LIN {X 0,Y 361.833,Z 229.413,A -85,B 0,C 180,E1 -13010.986,E2 -13010.986} C_VEL
LIN {X 0,Y 361.881,Z 229.41,A -85,B 0,C 180,E1 -13014.66,E2 -13014.66} C_VEL
LIN {X 0,Y 361.859,Z 229.412,A -85,B 0,C 180,E1 -13017.057,E2 -13017.057} C_VEL
LIN {X 0,Y 361.93,Z 229.564,A -85,B 0,C 180,E1 -13019.451,E2 -13019.451} C_VEL
LIN {X 0,Y 364.526,Z 241.261,A -85,B 0,C 180,E1 -13022.49,E2 -13022.49} C_VEL
LIN {X 0,Y 366.114,Z 250.204,A -85,B 0,C 180,E1 -13024.69,E2 -13024.69} C_VEL
LIN {X 0,Y 364.917,Z 262.619,A -85,B 0,C 180,E1 -13027.439,E2 -13027.439} C_VEL
LIN {X 0,Y 368.835,Z 283.762,A -85,B 0,C 180,E1 -13028.191,E2 -13028.191} C_VEL
LIN {X 0,Y 370.98,Z 298.524,A -85,B 0,C 180,E1 -13028.66,E2 -13028.66} C_VEL
LIN {X 0,Y 369.479,Z 372.16,A -85,B 0,C 180,E1 -13030.196,E2 -13030.196} C_VEL
LIN {X 0,Y 368.702,Z 385.754,A -85,B 0,C 180,E1 -13030.696,E2 -13030.696} C_VEL
LIN {X 0,Y 367.704,Z 398.62,A -85,B 0,C 180,E1 -13031.401,E2 -13031.401} C_VEL
LIN {X 0,Y 366.629,Z 410.378,A -85,B 0,C 180,E1 -13032.284,E2 -13032.284} C_VEL
LIN {X 0,Y 365.424,Z 421.749,A -85,B 0,C 180,E1 -13033.377,E2 -13033.377} C_VEL
LIN {X 0,Y 364.348,Z 431.632,A -85,B 0,C 180,E1 -13034.565,E2 -13034.565} C_VEL
LIN {X 0,Y 363.296,Z 441.299,A -85,B 0,C 180,E1 -13036.007,E2 -13036.007} C_VEL
LIN {X 0,Y 362.237,Z 450.344,A -85,B 0,C 180,E1 -13037.678,E2 -13037.678} C_VEL
LIN {X 0,Y 361.437,Z 457.643,A -85,B 0,C 180,E1 -13039.355,E2 -13039.355} C_VEL
LIN {X 0,Y 360.913,Z 463.485,A -85,B 0,C 180,E1 -13041.038,E2 -13041.038} C_VEL
LIN {X 0,Y 360.54,Z 468.095,A -85,B 0,C 180,E1 -13042.721,E2 -13042.721} C_VEL
LIN {X 0,Y 360.346,Z 471.611,A -85,B 0,C 180,E1 -13044.404,E2 -13044.404} C_VEL
LIN {X 0,Y 360.346,Z 473.371,A -85,B 0,C 180,E1 -13045.526,E2 -13045.526} C_VEL
LIN {X 0,Y 360.306,Z 474.719,A -85,B 0,C 180,E1 -13046.645,E2 -13046.645} C_VEL
LIN {X 0,Y 360.305,Z 475.671,A -85,B 0,C 180,E1 -13047.764,E2 -13047.764} C_VEL
LIN {X 0,Y 360.353,Z 476.208,A -85,B 0,C 180,E1 -13048.883,E2 -13048.883} C_VEL
LIN {X 0,Y 360.404,Z 476.312,A -85,B 0,C 180,E1 -13050,E2 -13050} C_VEL
LIN {X 0,Y 360.368,Z 476.021,A -85,B 0,C 180,E1 -13051.118,E2 -13051.118} C_VEL
LIN {X 0,Y 360.309,Z 475.335,A -85,B 0,C 180,E1 -13052.236,E2 -13052.236} C_VEL
LIN {X 0,Y 360.311,Z 474.232,A -85,B 0,C 180,E1 -13053.355,E2 -13053.355} C_VEL
LIN {X 0,Y 360.368,Z 472.675,A -85,B 0,C 180,E1 -13054.474,E2 -13054.474} C_VEL
LIN {X 0,Y 360.395,Z 469.967,A -85,B 0,C 180,E1 -13055.961,E2 -13055.961} C_VEL
LIN {X 0,Y 360.636,Z 465.301,A -85,B 0,C 180,E1 -13057.84,E2 -13057.84} C_VEL
LIN {X 0,Y 361.085,Z 458.852,A -85,B 0,C 180,E1 -13059.805,E2 -13059.805} C_VEL
LIN {X 0,Y 361.659,Z 451.801,A -85,B 0,C 180,E1 -13061.489,E2 -13061.489} C_VEL
LIN {X 0,Y 362.587,Z 442.961,A -85,B 0,C 180,E1 -13063.164,E2 -13063.164} C_VEL
LIN {X 0,Y 363.61,Z 432.861,A -85,B 0,C 180,E1 -13064.703,E2 -13064.703} C_VEL
LIN {X 0,Y 364.434,Z 422.644,A -85,B 0,C 180,E1 -13065.95,E2 -13065.95} C_VEL
LIN {X 0,Y 365.491,Z 411.272,A -85,B 0,C 180,E1 -13067.052,E2 -13067.052} C_VEL
LIN {X 0,Y 366.457,Z 399.49,A -85,B 0,C 180,E1 -13067.941,E2 -13067.941} C_VEL
LIN {X 0,Y 367.363,Z 386.617,A -85,B 0,C 180,E1 -13068.653,E2 -13068.653} C_VEL
LIN {X 0,Y 367.996,Z 374.094,A -85,B 0,C 180,E1 -13069.126,E2 -13069.126} C_VEL
LIN {X 0,Y 368.512,Z 346.999,A -85,B 0,C 180,E1 -13069.713,E2 -13069.713} C_VEL
LIN {X 0,Y 369.284,Z 296.844,A -85,B 0,C 180,E1 -13070.734,E2 -13070.734} C_VEL
LIN {X 0,Y 364.271,Z 263.791,A -85,B 0,C 180,E1 -13071.746,E2 -13071.746} C_VEL
LIN {X 0,Y 365.634,Z 249.234,A -85,B 0,C 180,E1 -13075.015,E2 -13075.015} C_VEL
LIN {X 0,Y 364.83,Z 243.927,A -85,B 0,C 180,E1 -13076.299,E2 -13076.299} C_VEL
LIN {X 0,Y 362.103,Z 230.432,A -85,B 0,C 180,E1 -13079.699,E2 -13079.699} C_VEL
LIN {X 0,Y 361.875,Z 229.413,A -85,B 0,C 180,E1 -13080.023,E2 -13080.023} C_VEL
LIN {X 0,Y 361.845,Z 229.41,A -85,B 0,C 180,E1 -13083.36,E2 -13083.36} C_VEL
LIN {X 0,Y 361.867,Z 229.406,A -85,B 0,C 180,E1 -13087.017,E2 -13087.017} C_VEL
LIN {X 0,Y 361.814,Z 229.412,A -85,B 0,C 180,E1 -13090.746,E2 -13090.746} C_VEL
LIN {X 0,Y 361.785,Z 229.417,A -85,B 0,C 180,E1 -13094.372,E2 -13094.372} C_VEL
LIN {X 0,Y 361.816,Z 229.417,A -85,B 0,C 180,E1 -13097.57,E2 -13097.57} C_VEL
LIN {X 0,Y 361.83,Z 229.411,A -85,B 0,C 180,E1 -13100.979,E2 -13100.979} C_VEL
LIN {X 0,Y 361.874,Z 229.405,A -85,B 0,C 180,E1 -13104.653,E2 -13104.653} C_VEL
LIN {X 0,Y 361.852,Z 229.408,A -85,B 0,C 180,E1 -13107.05,E2 -13107.05} C_VEL
LIN {X 0,Y 361.856,Z 229.408,A -85,B 0,C 180,E1 -13110.946,E2 -13110.946} C_VEL
LIN {X 0,Y 361.869,Z 229.405,A -85,B 0,C 180,E1 -13114.7,E2 -13114.7} C_VEL
LIN {X 0,Y 361.862,Z 229.407,A -85,B 0,C 180,E1 -13118.34,E2 -13118.34} C_VEL
LIN {X 0,Y 361.906,Z 229.403,A -85,B 0,C 180,E1 -13122.087,E2 -13122.087} C_VEL
LIN {X 0,Y 361.958,Z 229.398,A -85,B 0,C 180,E1 -13125.374,E2 -13125.374} C_VEL
LIN {X 0,Y 361.956,Z 229.395,A -85,B 0,C 180,E1 -13128.798,E2 -13128.798} C_VEL
LIN {X 0,Y 362.072,Z 229.381,A -85,B 0,C 180,E1 -13132.185,E2 -13132.185} C_VEL
LIN {X 0,Y 362.079,Z 229.379,A -85,B 0,C 180,E1 -13134.425,E2 -13134.425} C_VEL
LIN {X 0,Y 362.245,Z 229.362,A -85,B 0,C 180,E1 -13137.77,E2 -13137.77} C_VEL
LIN {X 0,Y 362.255,Z 229.358,A -85,B 0,C 180,E1 -13142.217,E2 -13142.217} C_VEL
LIN {X 0,Y 362.1,Z 229.377,A -85,B 0,C 180,E1 -13146.681,E2 -13146.681} C_VEL
LIN {X 0,Y 361.979,Z 229.393,A -85,B 0,C 180,E1 -13150.056,E2 -13150.056} C_VEL
LIN {X 0,Y 361.979,Z 229.394,A -85,B 0,C 180,E1 -13153.892,E2 -13153.892} C_VEL
LIN {X 0,Y 361.905,Z 229.403,A -85,B 0,C 180,E1 -13156.928,E2 -13156.928} C_VEL
LIN {X 0,Y 361.869,Z 229.405,A -85,B 0,C 180,E1 -13160.454,E2 -13160.454} C_VEL
LIN {X 0,Y 361.866,Z 229.406,A -85,B 0,C 180,E1 -13164.106,E2 -13164.106} C_VEL
LIN {X 0,Y 361.853,Z 229.41,A -85,B 0,C 180,E1 -13167.775,E2 -13167.775} C_VEL
LIN {X 0,Y 361.814,Z 229.418,A -85,B 0,C 180,E1 -13171.279,E2 -13171.279} C_VEL
LIN {X 0,Y 361.818,Z 229.412,A -85,B 0,C 180,E1 -13174.274,E2 -13174.274} C_VEL
LIN {X 0,Y 361.825,Z 229.416,A -85,B 0,C 180,E1 -13177.217,E2 -13177.217} C_VEL
LIN {X 0,Y 361.794,Z 229.416,A -85,B 0,C 180,E1 -13180.749,E2 -13180.749} C_VEL
LIN {X 0,Y 361.776,Z 229.417,A -85,B 0,C 180,E1 -13184.363,E2 -13184.363} C_VEL
LIN {X 0,Y 361.789,Z 229.419,A -85,B 0,C 180,E1 -13187.563,E2 -13187.563} C_VEL
LIN {X 0,Y 361.821,Z 229.415,A -85,B 0,C 180,E1 -13190.969,E2 -13190.969} C_VEL
LIN {X 0,Y 361.824,Z 229.412,A -85,B 0,C 180,E1 -13194.651,E2 -13194.651} C_VEL
LIN {X 0,Y 361.785,Z 229.416,A -85,B 0,C 180,E1 -13198.366,E2 -13198.366} C_VEL
LIN {X 0,Y 361.848,Z 229.412,A -85,B 0,C 180,E1 -13200.951,E2 -13200.951} C_VEL
LIN {X 0,Y 361.899,Z 229.405,A -85,B 0,C 180,E1 -13203.471,E2 -13203.471} C_VEL
LIN {X 0,Y 361.863,Z 229.413,A -85,B 0,C 180,E1 -13207.143,E2 -13207.143} C_VEL
LIN {X 0,Y 361.877,Z 229.407,A -85,B 0,C 180,E1 -13210.722,E2 -13210.722} C_VEL
LIN {X 0,Y 361.889,Z 229.403,A -85,B 0,C 180,E1 -13214.224,E2 -13214.224} C_VEL
LIN {X 0,Y 361.94,Z 229.398,A -85,B 0,C 180,E1 -13216.526,E2 -13216.526} C_VEL
LIN {X 0,Y 361.977,Z 229.392,A -85,B 0,C 180,E1 -13219.937,E2 -13219.937} C_VEL
LIN {X 0,Y 362.097,Z 229.377,A -85,B 0,C 180,E1 -13222.192,E2 -13222.192} C_VEL
LIN {X 0,Y 362.068,Z 229.381,A -85,B 0,C 180,E1 -13224.431,E2 -13224.431} C_VEL
LIN {X 0,Y 362.228,Z 229.361,A -85,B 0,C 180,E1 -13227.776,E2 -13227.776} C_VEL
LIN {X 0,Y 362.368,Z 229.343,A -85,B 0,C 180,E1 -13230,E2 -13230} C_VEL
LIN {X 0,Y 362.228,Z 229.361,A -85,B 0,C 180,E1 -13232.224,E2 -13232.224} C_VEL
LIN {X 0,Y 362.121,Z 229.377,A -85,B 0,C 180,E1 -13236.687,E2 -13236.687} C_VEL
LIN {X 0,Y 362.073,Z 229.567,A -85,B 0,C 180,E1 -13238.789,E2 -13238.789} C_VEL
LIN {X 0,Y 363.761,Z 238.743,A -85,B 0,C 180,E1 -13241.316,E2 -13241.316} C_VEL
LIN {X 0,Y 366.817,Z 248.552,A -85,B 0,C 180,E1 -13241.71,E2 -13241.71} C_VEL
LIN {X 0,Y 369.824,Z 264.217,A -85,B 0,C 180,E1 -13242.212,E2 -13242.212} C_VEL
LIN {X 0,Y 368.227,Z 346.682,A -85,B 0,C 180,E1 -13243.903,E2 -13243.903} C_VEL
LIN {X 0,Y 367.706,Z 359.685,A -85,B 0,C 180,E1 -13244.387,E2 -13244.387} C_VEL
LIN {X 0,Y 367.117,Z 371.772,A -85,B 0,C 180,E1 -13245.048,E2 -13245.048} C_VEL
LIN {X 0,Y 366.274,Z 384.403,A -85,B 0,C 180,E1 -13245.988,E2 -13245.988} C_VEL
LIN {X 0,Y 365.338,Z 395.535,A -85,B 0,C 180,E1 -13247.059,E2 -13247.059} C_VEL
LIN {X 0,Y 364.31,Z 406.448,A -85,B 0,C 180,E1 -13248.378,E2 -13248.378} C_VEL
LIN {X 0,Y 363.312,Z 415.93,A -85,B 0,C 180,E1 -13249.815,E2 -13249.815} C_VEL
LIN {X 0,Y 362.472,Z 424.801,A -85,B 0,C 180,E1 -13251.485,E2 -13251.485} C_VEL
LIN {X 0,Y 361.737,Z 431.855,A -85,B 0,C 180,E1 -13253.142,E2 -13253.142} C_VEL
LIN {X 0,Y 361.542,Z 433.936,A -85,B 0,C 180,E1 -13253.715,E2 -13253.715} C_VEL
LIN {X 0,Y 360.709,Z 436.714,A -85,B 0,C 180,E1 -13254.533,E2 -13254.533} C_VEL
LIN {X 0,Y 357.552,Z 440.748,A -85,B 0,C 180,E1 -13255.885,E2 -13255.885} C_VEL
LIN {X 0,Y 354.887,Z 443.525,A -85,B 0,C 180,E1 -13257.011,E2 -13257.011} C_VEL
LIN {X 0,Y 353.665,Z 445.304,A -85,B 0,C 180,E1 -13257.907,E2 -13257.907} C_VEL
LIN {X 0,Y 353.522,Z 445.8,A -85,B 0,C 180,E1 -13258.215,E2 -13258.215} C_VEL
LIN {X 0,Y 353.225,Z 448.061,A -85,B 0,C 180,E1 -13259.828,E2 -13259.828} C_VEL
LIN {X 0,Y 353.063,Z 449.259,A -85,B 0,C 180,E1 -13261.167,E2 -13261.167} C_VEL
LIN {X 0,Y 353.03,Z 450.068,A -85,B 0,C 180,E1 -13263.284,E2 -13263.284} C_VEL
LIN {X 0,Y 353.12,Z 449.518,A -85,B 0,C 180,E1 -13265.329,E2 -13265.329} C_VEL
LIN {X 0,Y 353.37,Z 447.743,A -85,B 0,C 180,E1 -13267.309,E2 -13267.309} C_VEL
LIN {X 0,Y 353.82,Z 444.396,A -85,B 0,C 180,E1 -13269.465,E2 -13269.465} C_VEL
LIN {X 0,Y 354.385,Z 439.268,A -85,B 0,C 180,E1 -13271.676,E2 -13271.676} C_VEL
LIN {X 0,Y 355.052,Z 434.218,A -85,B 0,C 180,E1 -13273.312,E2 -13273.312} C_VEL
LIN {X 0,Y 355.855,Z 428.017,A -85,B 0,C 180,E1 -13274.927,E2 -13274.927} C_VEL
LIN {X 0,Y 356.738,Z 421.001,A -85,B 0,C 180,E1 -13276.42,E2 -13276.42} C_VEL
LIN {X 0,Y 357.944,Z 411.554,A -85,B 0,C 180,E1 -13278.05,E2 -13278.05} C_VEL
LIN {X 0,Y 359.069,Z 402.36,A -85,B 0,C 180,E1 -13279.326,E2 -13279.326} C_VEL
LIN {X 0,Y 360.134,Z 392.431,A -85,B 0,C 180,E1 -13280.447,E2 -13280.447} C_VEL
LIN {X 0,Y 361.277,Z 380.527,A -85,B 0,C 180,E1 -13281.512,E2 -13281.512} C_VEL
LIN {X 0,Y 362.175,Z 368.681,A -85,B 0,C 180,E1 -13282.326,E2 -13282.326} C_VEL
LIN {X 0,Y 362.825,Z 356.306,A -85,B 0,C 180,E1 -13282.943,E2 -13282.943} C_VEL
LIN {X 0,Y 363.321,Z 342.566,A -85,B 0,C 180,E1 -13283.379,E2 -13283.379} C_VEL
LIN {X 0,Y 365.083,Z 265.657,A -85,B 0,C 180,E1 -13284.987,E2 -13284.987} C_VEL
LIN {X 0,Y 362.139,Z 252.353,A -85,B 0,C 180,E1 -13285.508,E2 -13285.508} C_VEL
LIN {X 0,Y 356.864,Z 239.401,A -85,B 0,C 180,E1 -13286.239,E2 -13286.239} C_VEL
LIN {X 0,Y 354.823,Z 230.291,A -85,B 0,C 180,E1 -13288.821,E2 -13288.821} C_VEL
LIN {X 0,Y 354.822,Z 230.288,A -85,B 0,C 180,E1 -13291.626,E2 -13291.626} C_VEL
LIN {X 0,Y 354.87,Z 230.279,A -85,B 0,C 180,E1 -13294.179,E2 -13294.179} C_VEL
LIN {X 0,Y 354.808,Z 230.287,A -85,B 0,C 180,E1 -13297.901,E2 -13297.901} C_VEL
LIN {X 0,Y 354.899,Z 230.279,A -85,B 0,C 180,E1 -13301.898,E2 -13301.898} C_VEL
LIN {X 0,Y 354.923,Z 230.272,A -85,B 0,C 180,E1 -13305.988,E2 -13305.988} C_VEL
LIN {X 0,Y 354.962,Z 230.269,A -85,B 0,C 180,E1 -13309.743,E2 -13309.743} C_VEL
LIN {X 0,Y 355.091,Z 230.254,A -85,B 0,C 180,E1 -13313.187,E2 -13313.187} C_VEL
LIN {X 0,Y 355.23,Z 230.231,A -85,B 0,C 180,E1 -13317.739,E2 -13317.739} C_VEL
LIN {X 0,Y 355.342,Z 230.22,A -85,B 0,C 180,E1 -13320.006,E2 -13320.006} C_VEL
LIN {X 0,Y 355.219,Z 230.23,A -85,B 0,C 180,E1 -13322.274,E2 -13322.274} C_VEL
LIN {X 0,Y 355.099,Z 230.248,A -85,B 0,C 180,E1 -13326.826,E2 -13326.826} C_VEL
LIN {X 0,Y 354.95,Z 230.263,A -85,B 0,C 180,E1 -13330.271,E2 -13330.271} C_VEL
LIN {X 0,Y 354.942,Z 230.266,A -85,B 0,C 180,E1 -13334.024,E2 -13334.024} C_VEL
LIN {X 0,Y 354.891,Z 230.273,A -85,B 0,C 180,E1 -13338.097,E2 -13338.097} C_VEL
LIN {X 0,Y 354.808,Z 230.284,A -85,B 0,C 180,E1 -13342.113,E2 -13342.113} C_VEL
LIN {X 0,Y 354.802,Z 230.285,A -85,B 0,C 180,E1 -13345.84,E2 -13345.84} C_VEL
LIN {X 0,Y 354.799,Z 230.285,A -85,B 0,C 180,E1 -13349.689,E2 -13349.689} C_VEL
LIN {X 0,Y 354.815,Z 230.281,A -85,B 0,C 180,E1 -13353.706,E2 -13353.706} C_VEL
LIN {X 0,Y 354.799,Z 230.287,A -85,B 0,C 180,E1 -13356.465,E2 -13356.465} C_VEL
LIN {X 0,Y 354.778,Z 230.289,A -85,B 0,C 180,E1 -13359.417,E2 -13359.417} C_VEL
LIN {X 0,Y 354.776,Z 230.295,A -85,B 0,C 180,E1 -13362.867,E2 -13362.867} C_VEL
LIN {X 0,Y 354.747,Z 230.302,A -85,B 0,C 180,E1 -13366.102,E2 -13366.102} C_VEL
LIN {X 0,Y 354.772,Z 230.293,A -85,B 0,C 180,E1 -13369.178,E2 -13369.178} C_VEL
LIN {X 0,Y 354.809,Z 230.289,A -85,B 0,C 180,E1 -13372.408,E2 -13372.408} C_VEL
LIN {X 0,Y 354.819,Z 230.288,A -85,B 0,C 180,E1 -13374.943,E2 -13374.943} C_VEL
LIN {X 0,Y 354.84,Z 230.387,A -85,B 0,C 180,E1 -13378.979,E2 -13378.979} C_VEL
LIN {X 0,Y 357.27,Z 241.039,A -85,B 0,C 180,E1 -13381.829,E2 -13381.829} C_VEL
LIN {X 0,Y 359.071,Z 250.386,A -85,B 0,C 180,E1 -13384.211,E2 -13384.211} C_VEL
LIN {X 0,Y 359.015,Z 254.237,A -85,B 0,C 180,E1 -13385.111,E2 -13385.111} C_VEL
LIN {X 0,Y 358.177,Z 262.294,A -85,B 0,C 180,E1 -13386.925,E2 -13386.925} C_VEL
LIN {X 0,Y 362.326,Z 284.308,A -85,B 0,C 180,E1 -13387.745,E2 -13387.745} C_VEL
LIN {X 0,Y 364.427,Z 299.076,A -85,B 0,C 180,E1 -13388.23,E2 -13388.23} C_VEL
LIN {X 0,Y 362.884,Z 372.032,A -85,B 0,C 180,E1 -13389.783,E2 -13389.783} C_VEL
LIN {X 0,Y 362.068,Z 385.57,A -85,B 0,C 180,E1 -13390.291,E2 -13390.291} C_VEL
LIN {X 0,Y 361.096,Z 397.89,A -85,B 0,C 180,E1 -13390.974,E2 -13390.974} C_VEL
LIN {X 0,Y 359.88,Z 410.544,A -85,B 0,C 180,E1 -13391.94,E2 -13391.94} C_VEL
LIN {X 0,Y 358.637,Z 421.837,A -85,B 0,C 180,E1 -13393.053,E2 -13393.053} C_VEL
LIN {X 0,Y 357.529,Z 431.546,A -85,B 0,C 180,E1 -13394.248,E2 -13394.248} C_VEL
LIN {X 0,Y 356.375,Z 441.257,A -85,B 0,C 180,E1 -13395.729,E2 -13395.729} C_VEL
LIN {X 0,Y 355.281,Z 450.253,A -85,B 0,C 180,E1 -13397.433,E2 -13397.433} C_VEL
LIN {X 0,Y 354.399,Z 457.509,A -85,B 0,C 180,E1 -13399.141,E2 -13399.141} C_VEL
LIN {X 0,Y 353.867,Z 463.313,A -85,B 0,C 180,E1 -13400.858,E2 -13400.858} C_VEL
LIN {X 0,Y 353.485,Z 467.901,A -85,B 0,C 180,E1 -13402.575,E2 -13402.575} C_VEL
LIN {X 0,Y 353.259,Z 471.4,A -85,B 0,C 180,E1 -13404.291,E2 -13404.291} C_VEL
LIN {X 0,Y 353.259,Z 473.149,A -85,B 0,C 180,E1 -13405.436,E2 -13405.436} C_VEL
LIN {X 0,Y 353.227,Z 474.49,A -85,B 0,C 180,E1 -13406.578,E2 -13406.578} C_VEL
LIN {X 0,Y 353.211,Z 475.432,A -85,B 0,C 180,E1 -13407.719,E2 -13407.719} C_VEL
LIN {X 0,Y 353.254,Z 475.95,A -85,B 0,C 180,E1 -13408.86,E2 -13408.86} C_VEL
LIN {X 0,Y 353.309,Z 476.044,A -85,B 0,C 180,E1 -13410,E2 -13410} C_VEL
LIN {X 0,Y 353.27,Z 475.742,A -85,B 0,C 180,E1 -13411.14,E2 -13411.14} C_VEL
LIN {X 0,Y 353.215,Z 475.047,A -85,B 0,C 180,E1 -13412.281,E2 -13412.281} C_VEL
LIN {X 0,Y 353.232,Z 473.922,A -85,B 0,C 180,E1 -13413.422,E2 -13413.422} C_VEL
LIN {X 0,Y 353.28,Z 472.353,A -85,B 0,C 180,E1 -13414.564,E2 -13414.564} C_VEL
LIN {X 0,Y 353.351,Z 469.184,A -85,B 0,C 180,E1 -13416.28,E2 -13416.28} C_VEL
LIN {X 0,Y 353.568,Z 464.928,A -85,B 0,C 180,E1 -13417.998,E2 -13417.998} C_VEL
LIN {X 0,Y 354.043,Z 458.448,A -85,B 0,C 180,E1 -13420.002,E2 -13420.002} C_VEL
LIN {X 0,Y 354.667,Z 451.351,A -85,B 0,C 180,E1 -13421.719,E2 -13421.719} C_VEL
LIN {X 0,Y 355.599,Z 442.465,A -85,B 0,C 180,E1 -13423.428,E2 -13423.428} C_VEL
LIN {X 0,Y 356.601,Z 433.359,A -85,B 0,C 180,E1 -13424.845,E2 -13424.845} C_VEL
LIN {X 0,Y 357.446,Z 423.303,A -85,B 0,C 180,E1 -13426.124,E2 -13426.124} C_VEL
LIN {X 0,Y 358.549,Z 412.143,A -85,B 0,C 180,E1 -13427.245,E2 -13427.245} C_VEL
LIN {X 0,Y 359.597,Z 399.65,A -85,B 0,C 180,E1 -13428.222,E2 -13428.222} C_VEL
LIN {X 0,Y 360.533,Z 386.995,A -85,B 0,C 180,E1 -13428.946,E2 -13428.946} C_VEL
LIN {X 0,Y 361.235,Z 373.669,A -85,B 0,C 180,E1 -13429.461,E2 -13429.461} C_VEL
LIN {X 0,Y 361.899,Z 341.43,A -85,B 0,C 180,E1 -13430.163,E2 -13430.163} C_VEL
LIN {X 0,Y 362.505,Z 297.423,A -85,B 0,C 180,E1 -13431.082,E2 -13431.082} C_VEL
LIN {X 0,Y 357.402,Z 263.613,A -85,B 0,C 180,E1 -13432.124,E2 -13432.124} C_VEL
LIN {X 0,Y 358.685,Z 250.088,A -85,B 0,C 180,E1 -13435.224,E2 -13435.224} C_VEL
LIN {X 0,Y 356.785,Z 239.68,A -85,B 0,C 180,E1 -13437.836,E2 -13437.836} C_VEL
LIN {X 0,Y 354.839,Z 230.287,A -85,B 0,C 180,E1 -13440.334,E2 -13440.334} C_VEL
LIN {X 0,Y 354.795,Z 230.292,A -85,B 0,C 180,E1 -13443.693,E2 -13443.693} C_VEL
LIN {X 0,Y 354.795,Z 230.287,A -85,B 0,C 180,E1 -13446.459,E2 -13446.459} C_VEL
LIN {X 0,Y 354.782,Z 230.291,A -85,B 0,C 180,E1 -13449.409,E2 -13449.409} C_VEL
LIN {X 0,Y 354.735,Z 230.294,A -85,B 0,C 180,E1 -13452.852,E2 -13452.852} C_VEL
LIN {X 0,Y 354.742,Z 230.296,A -85,B 0,C 180,E1 -13456.094,E2 -13456.094} C_VEL
LIN {X 0,Y 354.769,Z 230.291,A -85,B 0,C 180,E1 -13459.171,E2 -13459.171} C_VEL
LIN {X 0,Y 354.8,Z 230.287,A -85,B 0,C 180,E1 -13462.402,E2 -13462.402} C_VEL
LIN {X 0,Y 354.812,Z 230.285,A -85,B 0,C 180,E1 -13464.935,E2 -13464.935} C_VEL
LIN {X 0,Y 354.782,Z 230.289,A -85,B 0,C 180,E1 -13468.406,E2 -13468.406} C_VEL
LIN {X 0,Y 354.794,Z 230.293,A -85,B 0,C 180,E1 -13471.609,E2 -13471.609} C_VEL
LIN {X 0,Y 354.81,Z 230.289,A -85,B 0,C 180,E1 -13475.414,E2 -13475.414} C_VEL
LIN {X 0,Y 354.821,Z 230.285,A -85,B 0,C 180,E1 -13479.107,E2 -13479.107} C_VEL
LIN {X 0,Y 354.863,Z 230.278,A -85,B 0,C 180,E1 -13482.713,E2 -13482.713} C_VEL
LIN {X 0,Y 354.948,Z 230.268,A -85,B 0,C 180,E1 -13486.249,E2 -13486.249} C_VEL
LIN {X 0,Y 354.935,Z 230.274,A -85,B 0,C 180,E1 -13489.729,E2 -13489.729} C_VEL
LIN {X 0,Y 355.078,Z 230.254,A -85,B 0,C 180,E1 -13493.174,E2 -13493.174} C_VEL
LIN {X 0,Y 355.206,Z 230.24,A -85,B 0,C 180,E1 -13497.726,E2 -13497.726} C_VEL
LIN {X 0,Y 355.133,Z 230.247,A -85,B 0,C 180,E1 -13501.127,E2 -13501.127} C_VEL
LIN {X 0,Y 355.218,Z 230.234,A -85,B 0,C 180,E1 -13502.261,E2 -13502.261} C_VEL
LIN {X 0,Y 355.067,Z 230.253,A -85,B 0,C 180,E1 -13506.814,E2 -13506.814} C_VEL
LIN {X 0,Y 354.936,Z 230.269,A -85,B 0,C 180,E1 -13510.258,E2 -13510.258} C_VEL
LIN {X 0,Y 354.923,Z 230.272,A -85,B 0,C 180,E1 -13514.011,E2 -13514.011} C_VEL
LIN {X 0,Y 354.867,Z 230.278,A -85,B 0,C 180,E1 -13518.085,E2 -13518.085} C_VEL
LIN {X 0,Y 354.804,Z 230.286,A -85,B 0,C 180,E1 -13522.1,E2 -13522.1} C_VEL
LIN {X 0,Y 354.839,Z 230.283,A -85,B 0,C 180,E1 -13525.823,E2 -13525.823} C_VEL
LIN {X 0,Y 354.782,Z 230.291,A -85,B 0,C 180,E1 -13529.676,E2 -13529.676} C_VEL
LIN {X 0,Y 354.78,Z 230.291,A -85,B 0,C 180,E1 -13533.678,E2 -13533.678} C_VEL
LIN {X 0,Y 354.759,Z 230.291,A -85,B 0,C 180,E1 -13536.454,E2 -13536.454} C_VEL
LIN {X 0,Y 354.785,Z 230.293,A -85,B 0,C 180,E1 -13539.418,E2 -13539.418} C_VEL
LIN {X 0,Y 354.746,Z 230.295,A -85,B 0,C 180,E1 -13542.861,E2 -13542.861} C_VEL
LIN {X 0,Y 354.735,Z 230.294,A -85,B 0,C 180,E1 -13546.1,E2 -13546.1} C_VEL
LIN {X 0,Y 354.74,Z 230.299,A -85,B 0,C 180,E1 -13549.174,E2 -13549.174} C_VEL
LIN {X 0,Y 354.759,Z 230.291,A -85,B 0,C 180,E1 -13552.398,E2 -13552.398} C_VEL
LIN {X 0,Y 354.761,Z 230.294,A -85,B 0,C 180,E1 -13554.936,E2 -13554.936} C_VEL
LIN {X 0,Y 354.741,Z 230.294,A -85,B 0,C 180,E1 -13558.401,E2 -13558.401} C_VEL
LIN {X 0,Y 354.799,Z 230.288,A -85,B 0,C 180,E1 -13561.615,E2 -13561.615} C_VEL
LIN {X 0,Y 354.845,Z 230.28,A -85,B 0,C 180,E1 -13564.169,E2 -13564.169} C_VEL
LIN {X 0,Y 354.831,Z 230.283,A -85,B 0,C 180,E1 -13567.894,E2 -13567.894} C_VEL
LIN {X 0,Y 354.866,Z 230.278,A -85,B 0,C 180,E1 -13571.889,E2 -13571.889} C_VEL
LIN {X 0,Y 354.884,Z 230.276,A -85,B 0,C 180,E1 -13575.979,E2 -13575.979} C_VEL
LIN {X 0,Y 354.924,Z 230.271,A -85,B 0,C 180,E1 -13579.735,E2 -13579.735} C_VEL
LIN {X 0,Y 355.057,Z 230.254,A -85,B 0,C 180,E1 -13582.036,E2 -13582.036} C_VEL
LIN {X 0,Y 355.042,Z 230.256,A -85,B 0,C 180,E1 -13584.32,E2 -13584.32} C_VEL
LIN {X 0,Y 355.192,Z 230.238,A -85,B 0,C 180,E1 -13587.732,E2 -13587.732} C_VEL
LIN {X 0,Y 355.338,Z 230.219,A -85,B 0,C 180,E1 -13590,E2 -13590} C_VEL
LIN {X 0,Y 355.192,Z 230.237,A -85,B 0,C 180,E1 -13592.268,E2 -13592.268} C_VEL
LIN {X 0,Y 355.084,Z 230.255,A -85,B 0,C 180,E1 -13596.82,E2 -13596.82} C_VEL
LIN {X 0,Y 355.034,Z 230.331,A -85,B 0,C 180,E1 -13598.473,E2 -13598.473} C_VEL
LIN {X 0,Y 356.64,Z 239.192,A -85,B 0,C 180,E1 -13600.918,E2 -13600.918} C_VEL
LIN {X 0,Y 360.099,Z 249.495,A -85,B 0,C 180,E1 -13601.349,E2 -13601.349} C_VEL
LIN {X 0,Y 363.071,Z 264.63,A -85,B 0,C 180,E1 -13601.849,E2 -13601.849} C_VEL
LIN {X 0,Y 361.47,Z 346.947,A -85,B 0,C 180,E1 -13603.573,E2 -13603.573} C_VEL
LIN {X 0,Y 360.906,Z 360.062,A -85,B 0,C 180,E1 -13604.07,E2 -13604.07} C_VEL
LIN {X 0,Y 360.309,Z 372.372,A -85,B 0,C 180,E1 -13604.761,E2 -13604.761} C_VEL
LIN {X 0,Y 359.5,Z 383.509,A -85,B 0,C 180,E1 -13605.593,E2 -13605.593} C_VEL
LIN {X 0,Y 358.577,Z 394.778,A -85,B 0,C 180,E1 -13606.677,E2 -13606.677} C_VEL
LIN {X 0,Y 357.469,Z 406.034,A -85,B 0,C 180,E1 -13608.038,E2 -13608.038} C_VEL
LIN {X 0,Y 356.46,Z 415.155,A -85,B 0,C 180,E1 -13609.414,E2 -13609.414} C_VEL
LIN {X 0,Y 355.683,Z 422.848,A -85,B 0,C 180,E1 -13610.834,E2 -13610.834} C_VEL
LIN {X 0,Y 354.954,Z 429.845,A -85,B 0,C 180,E1 -13612.404,E2 -13612.404} C_VEL
LIN {X 0,Y 354.355,Z 436.249,A -85,B 0,C 180,E1 -13614.194,E2 -13614.194} C_VEL
LIN {X 0,Y 353.877,Z 441.074,A -85,B 0,C 180,E1 -13615.907,E2 -13615.907} C_VEL
LIN {X 0,Y 353.602,Z 445.19,A -85,B 0,C 180,E1 -13617.844,E2 -13617.844} C_VEL
LIN {X 0,Y 353.522,Z 445.8,A -85,B 0,C 180,E1 -13618.215,E2 -13618.215} C_VEL
LIN {X 0,Y 352.683,Z 447.239,A -85,B 0,C 180,E1 -13619.136,E2 -13619.136} C_VEL
LIN {X 0,Y 349.578,Z 449.014,A -85,B 0,C 180,E1 -13620.647,E2 -13620.647} C_VEL
LIN {X 0,Y 347.054,Z 449.897,A -85,B 0,C 180,E1 -13621.883,E2 -13621.883} C_VEL
LIN {X 0,Y 346.016,Z 450.252,A -85,B 0,C 180,E1 -13622.847,E2 -13622.847} C_VEL
LIN {X 0,Y 345.953,Z 450.296,A -85,B 0,C 180,E1 -13623.174,E2 -13623.174} C_VEL
LIN {X 0,Y 345.979,Z 450.116,A -85,B 0,C 180,E1 -13624.664,E2 -13624.664} C_VEL
LIN {X 0,Y 346.11,Z 449.345,A -85,B 0,C 180,E1 -13626.075,E2 -13626.075} C_VEL
LIN {X 0,Y 346.354,Z 447.689,A -85,B 0,C 180,E1 -13627.702,E2 -13627.702} C_VEL
LIN {X 0,Y 346.771,Z 444.651,A -85,B 0,C 180,E1 -13629.648,E2 -13629.648} C_VEL
LIN {X 0,Y 347.257,Z 440.523,A -85,B 0,C 180,E1 -13631.525,E2 -13631.525} C_VEL
LIN {X 0,Y 348.026,Z 435.115,A -85,B 0,C 180,E1 -13633.379,E2 -13633.379} C_VEL
LIN {X 0,Y 348.928,Z 428.381,A -85,B 0,C 180,E1 -13635.186,E2 -13635.186} C_VEL
LIN {X 0,Y 350.037,Z 420.084,A -85,B 0,C 180,E1 -13636.961,E2 -13636.961} C_VEL
LIN {X 0,Y 351.268,Z 411.04,A -85,B 0,C 180,E1 -13638.509,E2 -13638.509} C_VEL
LIN {X 0,Y 352.544,Z 400.844,A -85,B 0,C 180,E1 -13639.906,E2 -13639.906} C_VEL
LIN {X 0,Y 353.644,Z 390.683,A -85,B 0,C 180,E1 -13641.033,E2 -13641.033} C_VEL
LIN {X 0,Y 354.741,Z 379.626,A -85,B 0,C 180,E1 -13642.01,E2 -13642.01} C_VEL
LIN {X 0,Y 355.632,Z 367.858,A -85,B 0,C 180,E1 -13642.81,E2 -13642.81} C_VEL
LIN {X 0,Y 356.368,Z 354.697,A -85,B 0,C 180,E1 -13643.447,E2 -13643.447} C_VEL
LIN {X 0,Y 356.816,Z 341.333,A -85,B 0,C 180,E1 -13643.855,E2 -13643.855} C_VEL
LIN {X 0,Y 358.555,Z 266.365,A -85,B 0,C 180,E1 -13645.454,E2 -13645.454} C_VEL
LIN {X 0,Y 355.867,Z 254.347,A -85,B 0,C 180,E1 -13645.94,E2 -13645.94} C_VEL
LIN {X 0,Y 349.757,Z 239.716,A -85,B 0,C 180,E1 -13646.81,E2 -13646.81} C_VEL
LIN {X 0,Y 347.738,Z 231.172,A -85,B 0,C 180,E1 -13649.283,E2 -13649.283} C_VEL
LIN {X 0,Y 347.822,Z 231.159,A -85,B 0,C 180,E1 -13652.751,E2 -13652.751} C_VEL
LIN {X 0,Y 347.761,Z 231.166,A -85,B 0,C 180,E1 -13656.169,E2 -13656.169} C_VEL
LIN {X 0,Y 347.787,Z 231.163,A -85,B 0,C 180,E1 -13659.916,E2 -13659.916} C_VEL
LIN {X 0,Y 347.843,Z 231.157,A -85,B 0,C 180,E1 -13662.366,E2 -13662.366} C_VEL
LIN {X 0,Y 347.878,Z 231.15,A -85,B 0,C 180,E1 -13665.978,E2 -13665.978} C_VEL
LIN {X 0,Y 347.913,Z 231.148,A -85,B 0,C 180,E1 -13669.532,E2 -13669.532} C_VEL
LIN {X 0,Y 348.058,Z 231.131,A -85,B 0,C 180,E1 -13673.048,E2 -13673.048} C_VEL
LIN {X 0,Y 348.193,Z 231.108,A -85,B 0,C 180,E1 -13677.693,E2 -13677.693} C_VEL
LIN {X 0,Y 348.293,Z 231.098,A -85,B 0,C 180,E1 -13680.007,E2 -13680.007} C_VEL
LIN {X 0,Y 348.181,Z 231.107,A -85,B 0,C 180,E1 -13682.32,E2 -13682.32} C_VEL
LIN {X 0,Y 348.066,Z 231.125,A -85,B 0,C 180,E1 -13686.965,E2 -13686.965} C_VEL
LIN {X 0,Y 347.89,Z 231.143,A -85,B 0,C 180,E1 -13690.482,E2 -13690.482} C_VEL
LIN {X 0,Y 347.899,Z 231.142,A -85,B 0,C 180,E1 -13694.156,E2 -13694.156} C_VEL
LIN {X 0,Y 347.83,Z 231.152,A -85,B 0,C 180,E1 -13698.264,E2 -13698.264} C_VEL
LIN {X 0,Y 347.766,Z 231.161,A -85,B 0,C 180,E1 -13701.629,E2 -13701.629} C_VEL
LIN {X 0,Y 347.74,Z 231.165,A -85,B 0,C 180,E1 -13705.12,E2 -13705.12} C_VEL
LIN {X 0,Y 347.729,Z 231.167,A -85,B 0,C 180,E1 -13707.707,E2 -13707.707} C_VEL
LIN {X 0,Y 347.736,Z 231.164,A -85,B 0,C 180,E1 -13710.355,E2 -13710.355} C_VEL
LIN {X 0,Y 347.756,Z 231.161,A -85,B 0,C 180,E1 -13714.048,E2 -13714.048} C_VEL
LIN {X 0,Y 347.761,Z 231.163,A -85,B 0,C 180,E1 -13717.326,E2 -13717.326} C_VEL
LIN {X 0,Y 347.705,Z 231.173,A -85,B 0,C 180,E1 -13720.307,E2 -13720.307} C_VEL
LIN {X 0,Y 347.723,Z 231.174,A -85,B 0,C 180,E1 -13723.414,E2 -13723.414} C_VEL
LIN {X 0,Y 347.723,Z 231.174,A -85,B 0,C 180,E1 -13726.693,E2 -13726.693} C_VEL
LIN {X 0,Y 347.713,Z 231.178,A -85,B 0,C 180,E1 -13730.186,E2 -13730.186} C_VEL
LIN {X 0,Y 347.765,Z 231.167,A -85,B 0,C 180,E1 -13732.681,E2 -13732.681} C_VEL
LIN {X 0,Y 347.762,Z 231.172,A -85,B 0,C 180,E1 -13735.959,E2 -13735.959} C_VEL
LIN {X 0,Y 347.754,Z 231.184,A -85,B 0,C 180,E1 -13738.472,E2 -13738.472} C_VEL
LIN {X 0,Y 350.088,Z 241.049,A -85,B 0,C 180,E1 -13741.198,E2 -13741.198} C_VEL
LIN {X 0,Y 352.246,Z 252.287,A -85,B 0,C 180,E1 -13744.134,E2 -13744.134} C_VEL
LIN {X 0,Y 351.895,Z 258.179,A -85,B 0,C 180,E1 -13745.518,E2 -13745.518} C_VEL
LIN {X 0,Y 351.427,Z 261.974,A -85,B 0,C 180,E1 -13746.385,E2 -13746.385} C_VEL
LIN {X 0,Y 355.489,Z 283.186,A -85,B 0,C 180,E1 -13747.214,E2 -13747.214} C_VEL
LIN {X 0,Y 357.901,Z 299.559,A -85,B 0,C 180,E1 -13747.773,E2 -13747.773} C_VEL
LIN {X 0,Y 356.308,Z 371.996,A -85,B 0,C 180,E1 -13749.356,E2 -13749.356} C_VEL
LIN {X 0,Y 355.459,Z 385.426,A -85,B 0,C 180,E1 -13749.871,E2 -13749.871} C_VEL
LIN {X 0,Y 354.414,Z 398.188,A -85,B 0,C 180,E1 -13750.601,E2 -13750.601} C_VEL
LIN {X 0,Y 353.145,Z 410.71,A -85,B 0,C 180,E1 -13751.584,E2 -13751.584} C_VEL
LIN {X 0,Y 351.855,Z 421.925,A -85,B 0,C 180,E1 -13752.716,E2 -13752.716} C_VEL
LIN {X 0,Y 350.572,Z 432.426,A -85,B 0,C 180,E1 -13754.057,E2 -13754.057} C_VEL
LIN {X 0,Y 349.456,Z 441.216,A -85,B 0,C 180,E1 -13755.441,E2 -13755.441} C_VEL
LIN {X 0,Y 348.334,Z 450.178,A -85,B 0,C 180,E1 -13757.178,E2 -13757.178} C_VEL
LIN {X 0,Y 347.378,Z 457.393,A -85,B 0,C 180,E1 -13758.919,E2 -13758.919} C_VEL
LIN {X 0,Y 346.822,Z 463.162,A -85,B 0,C 180,E1 -13760.671,E2 -13760.671} C_VEL
LIN {X 0,Y 346.412,Z 467.721,A -85,B 0,C 180,E1 -13762.422,E2 -13762.422} C_VEL
LIN {X 0,Y 346.179,Z 471.194,A -85,B 0,C 180,E1 -13764.174,E2 -13764.174} C_VEL
LIN {X 0,Y 346.155,Z 472.931,A -85,B 0,C 180,E1 -13765.342,E2 -13765.342} C_VEL
LIN {X 0,Y 346.15,Z 474.262,A -85,B 0,C 180,E1 -13766.508,E2 -13766.508} C_VEL
LIN {X 0,Y 346.12,Z 475.193,A -85,B 0,C 180,E1 -13767.673,E2 -13767.673} C_VEL
LIN {X 0,Y 346.156,Z 475.691,A -85,B 0,C 180,E1 -13768.837,E2 -13768.837} C_VEL
LIN {X 0,Y 346.214,Z 475.776,A -85,B 0,C 180,E1 -13770,E2 -13770} C_VEL
LIN {X 0,Y 346.171,Z 475.464,A -85,B 0,C 180,E1 -13771.163,E2 -13771.163} C_VEL
LIN {X 0,Y 346.124,Z 474.758,A -85,B 0,C 180,E1 -13772.327,E2 -13772.327} C_VEL
LIN {X 0,Y 346.156,Z 473.613,A -85,B 0,C 180,E1 -13773.492,E2 -13773.492} C_VEL
LIN {X 0,Y 346.184,Z 470.716,A -85,B 0,C 180,E1 -13775.45,E2 -13775.45} C_VEL
LIN {X 0,Y 346.427,Z 466.116,A -85,B 0,C 180,E1 -13777.577,E2 -13777.577} C_VEL
LIN {X 0,Y 346.775,Z 461.055,A -85,B 0,C 180,E1 -13779.331,E2 -13779.331} C_VEL
LIN {X 0,Y 347.275,Z 454.676,A -85,B 0,C 180,E1 -13781.084,E2 -13781.084} C_VEL
LIN {X 0,Y 348.198,Z 446.68,A -85,B 0,C 180,E1 -13782.828,E2 -13782.828} C_VEL
LIN {X 0,Y 349.061,Z 438.515,A -85,B 0,C 180,E1 -13784.279,E2 -13784.279} C_VEL
LIN {X 0,Y 350.024,Z 428.98,A -85,B 0,C 180,E1 -13785.667,E2 -13785.667} C_VEL
LIN {X 0,Y 351.035,Z 418.755,A -85,B 0,C 180,E1 -13786.876,E2 -13786.876} C_VEL
LIN {X 0,Y 352.036,Z 408.16,A -85,B 0,C 180,E1 -13787.875,E2 -13787.875} C_VEL
LIN {X 0,Y 353.113,Z 395.437,A -85,B 0,C 180,E1 -13788.794,E2 -13788.794} C_VEL
LIN {X 0,Y 353.953,Z 382.763,A -85,B 0,C 180,E1 -13789.463,E2 -13789.463} C_VEL
LIN {X 0,Y 354.551,Z 369.312,A -85,B 0,C 180,E1 -13789.919,E2 -13789.919} C_VEL
LIN {X 0,Y 355.906,Z 299.314,A -85,B 0,C 180,E1 -13791.4,E2 -13791.4} C_VEL
LIN {X 0,Y 350.536,Z 263.319,A -85,B 0,C 180,E1 -13792.544,E2 -13792.544} C_VEL
LIN {X 0,Y 351.716,Z 251.169,A -85,B 0,C 180,E1 -13795.387,E2 -13795.387} C_VEL
LIN {X 0,Y 349.605,Z 239.846,A -85,B 0,C 180,E1 -13798.293,E2 -13798.293} C_VEL
LIN {X 0,Y 347.779,Z 231.164,A -85,B 0,C 180,E1 -13800.638,E2 -13800.638} C_VEL
LIN {X 0,Y 347.737,Z 231.167,A -85,B 0,C 180,E1 -13804.464,E2 -13804.464} C_VEL
LIN {X 0,Y 347.771,Z 231.166,A -85,B 0,C 180,E1 -13807.982,E2 -13807.982} C_VEL
LIN {X 0,Y 347.697,Z 231.176,A -85,B 0,C 180,E1 -13811.837,E2 -13811.837} C_VEL
LIN {X 0,Y 347.694,Z 231.172,A -85,B 0,C 180,E1 -13815.027,E2 -13815.027} C_VEL
LIN {X 0,Y 347.713,Z 231.17,A -85,B 0,C 180,E1 -13818.403,E2 -13818.403} C_VEL
LIN {X 0,Y 347.766,Z 231.165,A -85,B 0,C 180,E1 -13822.011,E2 -13822.011} C_VEL
LIN {X 0,Y 347.75,Z 231.169,A -85,B 0,C 180,E1 -13825.531,E2 -13825.531} C_VEL
LIN {X 0,Y 347.737,Z 231.167,A -85,B 0,C 180,E1 -13828.294,E2 -13828.294} C_VEL
LIN {X 0,Y 347.739,Z 231.166,A -85,B 0,C 180,E1 -13830.978,E2 -13830.978} C_VEL
LIN {X 0,Y 347.74,Z 231.171,A -85,B 0,C 180,E1 -13833.595,E2 -13833.595} C_VEL
LIN {X 0,Y 347.755,Z 231.165,A -85,B 0,C 180,E1 -13836.154,E2 -13836.154} C_VEL
LIN {X 0,Y 347.769,Z 231.165,A -85,B 0,C 180,E1 -13839.901,E2 -13839.901} C_VEL
LIN {X 0,Y 347.82,Z 231.162,A -85,B 0,C 180,E1 -13843.562,E2 -13843.562} C_VEL
LIN {X 0,Y 347.883,Z 231.15,A -85,B 0,C 180,E1 -13847.154,E2 -13847.154} C_VEL
LIN {X 0,Y 347.925,Z 231.143,A -85,B 0,C 180,E1 -13850.694,E2 -13850.694} C_VEL
LIN {X 0,Y 348.028,Z 231.13,A -85,B 0,C 180,E1 -13854.199,E2 -13854.199} C_VEL
LIN {X 0,Y 348.144,Z 231.12,A -85,B 0,C 180,E1 -13857.68,E2 -13857.68} C_VEL
LIN {X 0,Y 348.105,Z 231.123,A -85,B 0,C 180,E1 -13861.15,E2 -13861.15} C_VEL
LIN {X 0,Y 348.179,Z 231.111,A -85,B 0,C 180,E1 -13862.307,E2 -13862.307} C_VEL
LIN {X 0,Y 348.034,Z 231.13,A -85,B 0,C 180,E1 -13866.952,E2 -13866.952} C_VEL
LIN {X 0,Y 347.876,Z 231.149,A -85,B 0,C 180,E1 -13870.469,E2 -13870.469} C_VEL
LIN {X 0,Y 347.88,Z 231.149,A -85,B 0,C 180,E1 -13874.143,E2 -13874.143} C_VEL
LIN {X 0,Y 347.807,Z 231.157,A -85,B 0,C 180,E1 -13878.252,E2 -13878.252} C_VEL
LIN {X 0,Y 347.761,Z 231.167,A -85,B 0,C 180,E1 -13881.627,E2 -13881.627} C_VEL
LIN {X 0,Y 347.767,Z 231.165,A -85,B 0,C 180,E1 -13885.103,E2 -13885.103} C_VEL
LIN {X 0,Y 347.759,Z 231.166,A -85,B 0,C 180,E1 -13887.689,E2 -13887.689} C_VEL
LIN {X 0,Y 347.714,Z 231.169,A -85,B 0,C 180,E1 -13890.342,E2 -13890.342} C_VEL
LIN {X 0,Y 347.713,Z 231.169,A -85,B 0,C 180,E1 -13894.037,E2 -13894.037} C_VEL
LIN {X 0,Y 347.723,Z 231.174,A -85,B 0,C 180,E1 -13897.315,E2 -13897.315} C_VEL
LIN {X 0,Y 347.692,Z 231.171,A -85,B 0,C 180,E1 -13900.291,E2 -13900.291} C_VEL
LIN {X 0,Y 347.681,Z 231.178,A -85,B 0,C 180,E1 -13903.402,E2 -13903.402} C_VEL
LIN {X 0,Y 347.683,Z 231.174,A -85,B 0,C 180,E1 -13906.68,E2 -13906.68} C_VEL
LIN {X 0,Y 347.7,Z 231.17,A -85,B 0,C 180,E1 -13910.168,E2 -13910.168} C_VEL
LIN {X 0,Y 347.713,Z 231.17,A -85,B 0,C 180,E1 -13912.674,E2 -13912.674} C_VEL
LIN {X 0,Y 347.698,Z 231.171,A -85,B 0,C 180,E1 -13915.952,E2 -13915.952} C_VEL
LIN {X 0,Y 347.712,Z 231.171,A -85,B 0,C 180,E1 -13919.649,E2 -13919.649} C_VEL
LIN {X 0,Y 347.799,Z 231.16,A -85,B 0,C 180,E1 -13922.741,E2 -13922.741} C_VEL
LIN {X 0,Y 347.76,Z 231.163,A -85,B 0,C 180,E1 -13926.16,E2 -13926.16} C_VEL
LIN {X 0,Y 347.782,Z 231.161,A -85,B 0,C 180,E1 -13929.908,E2 -13929.908} C_VEL
LIN {X 0,Y 347.81,Z 231.157,A -85,B 0,C 180,E1 -13932.357,E2 -13932.357} C_VEL
LIN {X 0,Y 347.84,Z 231.153,A -85,B 0,C 180,E1 -13935.969,E2 -13935.969} C_VEL
LIN {X 0,Y 347.874,Z 231.151,A -85,B 0,C 180,E1 -13939.524,E2 -13939.524} C_VEL
LIN {X 0,Y 348.017,Z 231.131,A -85,B 0,C 180,E1 -13941.874,E2 -13941.874} C_VEL
LIN {X 0,Y 348.017,Z 231.131,A -85,B 0,C 180,E1 -13944.205,E2 -13944.205} C_VEL
LIN {X 0,Y 348.155,Z 231.115,A -85,B 0,C 180,E1 -13947.686,E2 -13947.686} C_VEL
LIN {X 0,Y 348.308,Z 231.095,A -85,B 0,C 180,E1 -13950,E2 -13950} C_VEL
LIN {X 0,Y 348.155,Z 231.114,A -85,B 0,C 180,E1 -13952.314,E2 -13952.314} C_VEL
LIN {X 0,Y 348.05,Z 231.133,A -85,B 0,C 180,E1 -13956.958,E2 -13956.958} C_VEL
LIN {X 0,Y 348.038,Z 231.285,A -85,B 0,C 180,E1 -13958.199,E2 -13958.199} C_VEL
LIN {X 0,Y 349.457,Z 239.196,A -85,B 0,C 180,E1 -13960.464,E2 -13960.464} C_VEL
LIN {X 0,Y 353.77,Z 252.171,A -85,B 0,C 180,E1 -13961.041,E2 -13961.041} C_VEL
LIN {X 0,Y 356.397,Z 266.186,A -85,B 0,C 180,E1 -13961.508,E2 -13961.508} C_VEL
LIN {X 0,Y 354.731,Z 346.581,A -85,B 0,C 180,E1 -13963.217,E2 -13963.217} C_VEL
LIN {X 0,Y 354.14,Z 359.706,A -85,B 0,C 180,E1 -13963.713,E2 -13963.713} C_VEL
LIN {X 0,Y 353.476,Z 372.905,A -85,B 0,C 180,E1 -13964.464,E2 -13964.464} C_VEL
LIN {X 0,Y 352.656,Z 383.952,A -85,B 0,C 180,E1 -13965.31,E2 -13965.31} C_VEL
LIN {X 0,Y 351.662,Z 395.43,A -85,B 0,C 180,E1 -13966.441,E2 -13966.441} C_VEL
LIN {X 0,Y 350.545,Z 406.434,A -85,B 0,C 180,E1 -13967.802,E2 -13967.802} C_VEL
LIN {X 0,Y 349.474,Z 415.702,A -85,B 0,C 180,E1 -13969.236,E2 -13969.236} C_VEL
LIN {X 0,Y 348.537,Z 424.705,A -85,B 0,C 180,E1 -13970.972,E2 -13970.972} C_VEL
LIN {X 0,Y 347.67,Z 432.64,A -85,B 0,C 180,E1 -13972.9,E2 -13972.9} C_VEL
LIN {X 0,Y 347.045,Z 438.522,A -85,B 0,C 180,E1 -13974.733,E2 -13974.733} C_VEL
LIN {X 0,Y 346.644,Z 443.766,A -85,B 0,C 180,E1 -13976.886,E2 -13976.886} C_VEL
LIN {X 0,Y 346.378,Z 446.572,A -85,B 0,C 180,E1 -13978.477,E2 -13978.477} C_VEL
LIN {X 0,Y 346.025,Z 449.026,A -85,B 0,C 180,E1 -13980.514,E2 -13980.514} C_VEL
LIN {X 0,Y 345.947,Z 449.936,A -85,B 0,C 180,E1 -13981.883,E2 -13981.883} C_VEL
LIN {X 0,Y 345.953,Z 450.296,A -85,B 0,C 180,E1 -13983.174,E2 -13983.174} C_VEL
LIN {X 0,Y 345.351,Z 450.406,A -85,B 0,C 180,E1 -13984.147,E2 -13984.147} C_VEL
LIN {X 0,Y 342.589,Z 449.909,A -85,B 0,C 180,E1 -13985.732,E2 -13985.732} C_VEL
LIN {X 0,Y 340.287,Z 448.907,A -85,B 0,C 180,E1 -13987.006,E2 -13987.006} C_VEL
LIN {X 0,Y 339.387,Z 447.8,A -85,B 0,C 180,E1 -13987.981,E2 -13987.981} C_VEL
LIN {X 0,Y 339.363,Z 447.364,A -85,B 0,C 180,E1 -13988.308,E2 -13988.308} C_VEL
LIN {X 0,Y 339.791,Z 444.46,A -85,B 0,C 180,E1 -13990.082,E2 -13990.082} C_VEL
LIN {X 0,Y 340.345,Z 440.153,A -85,B 0,C 180,E1 -13991.993,E2 -13991.993} C_VEL
LIN {X 0,Y 341.168,Z 434.577,A -85,B 0,C 180,E1 -13993.877,E2 -13993.877} C_VEL
LIN {X 0,Y 342.19,Z 427.645,A -85,B 0,C 180,E1 -13995.722,E2 -13995.722} C_VEL
LIN {X 0,Y 343.354,Z 419.468,A -85,B 0,C 180,E1 -13997.464,E2 -13997.464} C_VEL
LIN {X 0,Y 344.596,Z 410.521,A -85,B 0,C 180,E1 -13998.989,E2 -13998.989} C_VEL
LIN {X 0,Y 345.885,Z 400.696,A -85,B 0,C 180,E1 -14000.347,E2 -14000.347} C_VEL
LIN {X 0,Y 347.218,Z 389.106,A -85,B 0,C 180,E1 -14001.629,E2 -14001.629} C_VEL
LIN {X 0,Y 348.417,Z 376.328,A -85,B 0,C 180,E1 -14002.707,E2 -14002.707} C_VEL
LIN {X 0,Y 349.376,Z 363.771,A -85,B 0,C 180,E1 -14003.494,E2 -14003.494} C_VEL
LIN {X 0,Y 350.056,Z 350.642,A -85,B 0,C 180,E1 -14004.056,E2 -14004.056} C_VEL
LIN {X 0,Y 350.587,Z 331.74,A -85,B 0,C 180,E1 -14004.523,E2 -14004.523} C_VEL
LIN {X 0,Y 352.189,Z 267.716,A -85,B 0,C 180,E1 -14005.912,E2 -14005.912} C_VEL
LIN {X 0,Y 349.884,Z 257.216,A -85,B 0,C 180,E1 -14006.35,E2 -14006.35} C_VEL
LIN {X 0,Y 342.624,Z 240.105,A -85,B 0,C 180,E1 -14007.394,E2 -14007.394} C_VEL
LIN {X 0,Y 340.718,Z 232.046,A -85,B 0,C 180,E1 -14009.777,E2 -14009.777} C_VEL
LIN {X 0,Y 340.775,Z 232.039,A -85,B 0,C 180,E1 -14013.027,E2 -14013.027} C_VEL
LIN {X 0,Y 340.701,Z 232.051,A -85,B 0,C 180,E1 -14016.934,E2 -14016.934} C_VEL
LIN {X 0,Y 340.767,Z 232.039,A -85,B 0,C 180,E1 -14020.74,E2 -14020.74} C_VEL
LIN {X 0,Y 340.764,Z 232.039,A -85,B 0,C 180,E1 -14023.226,E2 -14023.226} C_VEL
LIN {X 0,Y 340.828,Z 232.034,A -85,B 0,C 180,E1 -14026.897,E2 -14026.897} C_VEL
LIN {X 0,Y 340.896,Z 232.023,A -85,B 0,C 180,E1 -14030.514,E2 -14030.514} C_VEL
LIN {X 0,Y 341.027,Z 232.007,A -85,B 0,C 180,E1 -14032.904,E2 -14032.904} C_VEL
LIN {X 0,Y 341.154,Z 231.985,A -85,B 0,C 180,E1 -14037.645,E2 -14037.645} C_VEL
LIN {X 0,Y 341.245,Z 231.976,A -85,B 0,C 180,E1 -14040.007,E2 -14040.007} C_VEL
LIN {X 0,Y 341.119,Z 231.986,A -85,B 0,C 180,E1 -14042.368,E2 -14042.368} C_VEL
LIN {X 0,Y 341.035,Z 232.002,A -85,B 0,C 180,E1 -14047.109,E2 -14047.109} C_VEL
LIN {X 0,Y 340.843,Z 232.022,A -85,B 0,C 180,E1 -14050.701,E2 -14050.701} C_VEL
LIN {X 0,Y 340.863,Z 232.018,A -85,B 0,C 180,E1 -14054.331,E2 -14054.331} C_VEL
LIN {X 0,Y 340.787,Z 232.028,A -85,B 0,C 180,E1 -14058.446,E2 -14058.446} C_VEL
LIN {X 0,Y 340.722,Z 232.039,A -85,B 0,C 180,E1 -14061.847,E2 -14061.847} C_VEL
LIN {X 0,Y 340.674,Z 232.045,A -85,B 0,C 180,E1 -14065.678,E2 -14065.678} C_VEL
LIN {X 0,Y 340.68,Z 232.049,A -85,B 0,C 180,E1 -14068.331,E2 -14068.331} C_VEL
LIN {X 0,Y 340.689,Z 232.046,A -85,B 0,C 180,E1 -14071.051,E2 -14071.051} C_VEL
LIN {X 0,Y 340.723,Z 232.042,A -85,B 0,C 180,E1 -14075.284,E2 -14075.284} C_VEL
LIN {X 0,Y 340.701,Z 232.049,A -85,B 0,C 180,E1 -14078.386,E2 -14078.386} C_VEL
LIN {X 0,Y 340.674,Z 232.051,A -85,B 0,C 180,E1 -14082.043,E2 -14082.043} C_VEL
LIN {X 0,Y 340.637,Z 232.056,A -85,B 0,C 180,E1 -14085.455,E2 -14085.455} C_VEL
LIN {X 0,Y 340.655,Z 232.054,A -85,B 0,C 180,E1 -14088.687,E2 -14088.687} C_VEL
LIN {X 0,Y 340.73,Z 232.044,A -85,B 0,C 180,E1 -14091.773,E2 -14091.773} C_VEL
LIN {X 0,Y 340.736,Z 232.044,A -85,B 0,C 180,E1 -14095.599,E2 -14095.599} C_VEL
LIN {X 0,Y 340.726,Z 232.156,A -85,B 0,C 180,E1 -14097.98,E2 -14097.98} C_VEL
LIN {X 0,Y 343.136,Z 242.234,A -85,B 0,C 180,E1 -14100.856,E2 -14100.856} C_VEL
LIN {X 0,Y 345.339,Z 253.379,A -85,B 0,C 180,E1 -14103.845,E2 -14103.845} C_VEL
LIN {X 0,Y 345.171,Z 258.179,A -85,B 0,C 180,E1 -14105.009,E2 -14105.009} C_VEL
LIN {X 0,Y 344.773,Z 261.637,A -85,B 0,C 180,E1 -14105.821,E2 -14105.821} C_VEL
LIN {X 0,Y 349.168,Z 284.713,A -85,B 0,C 180,E1 -14106.761,E2 -14106.761} C_VEL
LIN {X 0,Y 351.495,Z 300.865,A -85,B 0,C 180,E1 -14107.326,E2 -14107.326} C_VEL
LIN {X 0,Y 349.845,Z 371.063,A -85,B 0,C 180,E1 -14108.879,E2 -14108.879} C_VEL
LIN {X 0,Y 348.948,Z 384.699,A -85,B 0,C 180,E1 -14109.401,E2 -14109.401} C_VEL
LIN {X 0,Y 347.854,Z 397.607,A -85,B 0,C 180,E1 -14110.143,E2 -14110.143} C_VEL
LIN {X 0,Y 346.633,Z 409.385,A -85,B 0,C 180,E1 -14111.071,E2 -14111.071} C_VEL
LIN {X 0,Y 345.216,Z 420.772,A -85,B 0,C 180,E1 -14112.22,E2 -14112.22} C_VEL
LIN {X 0,Y 344.043,Z 430.008,A -85,B 0,C 180,E1 -14113.383,E2 -14113.383} C_VEL
LIN {X 0,Y 342.821,Z 439.529,A -85,B 0,C 180,E1 -14114.848,E2 -14114.848} C_VEL
LIN {X 0,Y 341.591,Z 448.731,A -85,B 0,C 180,E1 -14116.617,E2 -14116.617} C_VEL
LIN {X 0,Y 340.49,Z 456.165,A -85,B 0,C 180,E1 -14118.39,E2 -14118.39} C_VEL
LIN {X 0,Y 339.957,Z 461.225,A -85,B 0,C 180,E1 -14119.88,E2 -14119.88} C_VEL
LIN {X 0,Y 339.477,Z 466.15,A -85,B 0,C 180,E1 -14121.668,E2 -14121.668} C_VEL
LIN {X 0,Y 339.174,Z 469.947,A -85,B 0,C 180,E1 -14123.456,E2 -14123.456} C_VEL
LIN {X 0,Y 339.057,Z 472.72,A -85,B 0,C 180,E1 -14125.244,E2 -14125.244} C_VEL
LIN {X 0,Y 339.073,Z 474.04,A -85,B 0,C 180,E1 -14126.435,E2 -14126.435} C_VEL
LIN {X 0,Y 339.032,Z 474.957,A -85,B 0,C 180,E1 -14127.624,E2 -14127.624} C_VEL
LIN {X 0,Y 339.058,Z 475.433,A -85,B 0,C 180,E1 -14128.812,E2 -14128.812} C_VEL
LIN {X 0,Y 339.118,Z 475.506,A -85,B 0,C 180,E1 -14130,E2 -14130} C_VEL
LIN {X 0,Y 339.073,Z 475.182,A -85,B 0,C 180,E1 -14131.188,E2 -14131.188} C_VEL
LIN {X 0,Y 339.036,Z 474.463,A -85,B 0,C 180,E1 -14132.376,E2 -14132.376} C_VEL
LIN {X 0,Y 339.082,Z 473.294,A -85,B 0,C 180,E1 -14133.565,E2 -14133.565} C_VEL
LIN {X 0,Y 339.128,Z 469.856,A -85,B 0,C 180,E1 -14135.848,E2 -14135.848} C_VEL
LIN {X 0,Y 339.369,Z 465.739,A -85,B 0,C 180,E1 -14137.736,E2 -14137.736} C_VEL
LIN {X 0,Y 339.817,Z 459.657,A -85,B 0,C 180,E1 -14139.824,E2 -14139.824} C_VEL
LIN {X 0,Y 340.388,Z 452.962,A -85,B 0,C 180,E1 -14141.613,E2 -14141.613} C_VEL
LIN {X 0,Y 341.407,Z 444.655,A -85,B 0,C 180,E1 -14143.39,E2 -14143.39} C_VEL
LIN {X 0,Y 342.435,Z 435.284,A -85,B 0,C 180,E1 -14144.997,E2 -14144.997} C_VEL
LIN {X 0,Y 343.482,Z 424.391,A -85,B 0,C 180,E1 -14146.493,E2 -14146.493} C_VEL
LIN {X 0,Y 344.61,Z 413.711,A -85,B 0,C 180,E1 -14147.659,E2 -14147.659} C_VEL
LIN {X 0,Y 345.744,Z 401.786,A -85,B 0,C 180,E1 -14148.672,E2 -14148.672} C_VEL
LIN {X 0,Y 346.728,Z 389.423,A -85,B 0,C 180,E1 -14149.461,E2 -14149.461} C_VEL
LIN {X 0,Y 347.494,Z 376.8,A -85,B 0,C 180,E1 -14150.032,E2 -14150.032} C_VEL
LIN {X 0,Y 347.989,Z 362.112,A -85,B 0,C 180,E1 -14150.426,E2 -14150.426} C_VEL
LIN {X 0,Y 349.118,Z 299.105,A -85,B 0,C 180,E1 -14151.784,E2 -14151.784} C_VEL
LIN {X 0,Y 343.661,Z 263.082,A -85,B 0,C 180,E1 -14152.964,E2 -14152.964} C_VEL
LIN {X 0,Y 344.745,Z 253.078,A -85,B 0,C 180,E1 -14155.347,E2 -14155.347} C_VEL
LIN {X 0,Y 343.441,Z 245.096,A -85,B 0,C 180,E1 -14157.414,E2 -14157.414} C_VEL
LIN {X 0,Y 340.854,Z 232.679,A -85,B 0,C 180,E1 -14160.77,E2 -14160.77} C_VEL
LIN {X 0,Y 340.716,Z 232.043,A -85,B 0,C 180,E1 -14160.977,E2 -14160.977} C_VEL
LIN {X 0,Y 340.716,Z 232.042,A -85,B 0,C 180,E1 -14165.278,E2 -14165.278} C_VEL
LIN {X 0,Y 340.704,Z 232.043,A -85,B 0,C 180,E1 -14168.378,E2 -14168.378} C_VEL
LIN {X 0,Y 340.638,Z 232.054,A -85,B 0,C 180,E1 -14172.028,E2 -14172.028} C_VEL
LIN {X 0,Y 340.634,Z 232.054,A -85,B 0,C 180,E1 -14175.447,E2 -14175.447} C_VEL
LIN {X 0,Y 340.651,Z 232.049,A -85,B 0,C 180,E1 -14178.679,E2 -14178.679} C_VEL
LIN {X 0,Y 340.724,Z 232.045,A -85,B 0,C 180,E1 -14181.766,E2 -14181.766} C_VEL
LIN {X 0,Y 340.73,Z 232.044,A -85,B 0,C 180,E1 -14185.592,E2 -14185.592} C_VEL
LIN {X 0,Y 340.688,Z 232.044,A -85,B 0,C 180,E1 -14188.949,E2 -14188.949} C_VEL
LIN {X 0,Y 340.715,Z 232.041,A -85,B 0,C 180,E1 -14193.007,E2 -14193.007} C_VEL
LIN {X 0,Y 340.708,Z 232.042,A -85,B 0,C 180,E1 -14196.92,E2 -14196.92} C_VEL
LIN {X 0,Y 340.703,Z 232.042,A -85,B 0,C 180,E1 -14200.722,E2 -14200.722} C_VEL
LIN {X 0,Y 340.811,Z 232.029,A -85,B 0,C 180,E1 -14204.444,E2 -14204.444} C_VEL
LIN {X 0,Y 340.84,Z 232.026,A -85,B 0,C 180,E1 -14208.094,E2 -14208.094} C_VEL
LIN {X 0,Y 340.977,Z 232.013,A -85,B 0,C 180,E1 -14211.698,E2 -14211.698} C_VEL
LIN {X 0,Y 341.004,Z 232.006,A -85,B 0,C 180,E1 -14214.079,E2 -14214.079} C_VEL
LIN {X 0,Y 341.085,Z 232,A -85,B 0,C 180,E1 -14217.632,E2 -14217.632} C_VEL
LIN {X 0,Y 341.076,Z 231.998,A -85,B 0,C 180,E1 -14221.174,E2 -14221.174} C_VEL
LIN {X 0,Y 341.116,Z 231.991,A -85,B 0,C 180,E1 -14222.355,E2 -14222.355} C_VEL
LIN {X 0,Y 340.982,Z 232.01,A -85,B 0,C 180,E1 -14227.097,E2 -14227.097} C_VEL
LIN {X 0,Y 340.828,Z 232.027,A -85,B 0,C 180,E1 -14230.688,E2 -14230.688} C_VEL
LIN {X 0,Y 340.844,Z 232.025,A -85,B 0,C 180,E1 -14234.318,E2 -14234.318} C_VEL
LIN {X 0,Y 340.764,Z 232.035,A -85,B 0,C 180,E1 -14238.433,E2 -14238.433} C_VEL
LIN {X 0,Y 340.729,Z 232.041,A -85,B 0,C 180,E1 -14241.85,E2 -14241.85} C_VEL
LIN {X 0,Y 340.723,Z 232.043,A -85,B 0,C 180,E1 -14245.659,E2 -14245.659} C_VEL
LIN {X 0,Y 340.687,Z 232.044,A -85,B 0,C 180,E1 -14248.315,E2 -14248.315} C_VEL
LIN {X 0,Y 340.664,Z 232.05,A -85,B 0,C 180,E1 -14251.038,E2 -14251.038} C_VEL
LIN {X 0,Y 340.681,Z 232.051,A -85,B 0,C 180,E1 -14255.273,E2 -14255.273} C_VEL
LIN {X 0,Y 340.671,Z 232.046,A -85,B 0,C 180,E1 -14258.379,E2 -14258.379} C_VEL
LIN {X 0,Y 340.658,Z 232.048,A -85,B 0,C 180,E1 -14262.039,E2 -14262.039} C_VEL
LIN {X 0,Y 340.641,Z 232.054,A -85,B 0,C 180,E1 -14265.456,E2 -14265.456} C_VEL
LIN {X 0,Y 340.639,Z 232.051,A -85,B 0,C 180,E1 -14268.685,E2 -14268.685} C_VEL
LIN {X 0,Y 340.685,Z 232.046,A -85,B 0,C 180,E1 -14271.767,E2 -14271.767} C_VEL
LIN {X 0,Y 340.673,Z 232.048,A -85,B 0,C 180,E1 -14275.591,E2 -14275.591} C_VEL
LIN {X 0,Y 340.652,Z 232.052,A -85,B 0,C 180,E1 -14278.952,E2 -14278.952} C_VEL
LIN {X 0,Y 340.726,Z 232.04,A -85,B 0,C 180,E1 -14282.47,E2 -14282.47} C_VEL
LIN {X 0,Y 340.736,Z 232.04,A -85,B 0,C 180,E1 -14285.637,E2 -14285.637} C_VEL
LIN {X 0,Y 340.726,Z 232.042,A -85,B 0,C 180,E1 -14289.473,E2 -14289.473} C_VEL
LIN {X 0,Y 340.802,Z 232.03,A -85,B 0,C 180,E1 -14291.982,E2 -14291.982} C_VEL
LIN {X 0,Y 340.812,Z 232.03,A -85,B 0,C 180,E1 -14295.703,E2 -14295.703} C_VEL
LIN {X 0,Y 340.816,Z 232.032,A -85,B 0,C 180,E1 -14299.305,E2 -14299.305} C_VEL
LIN {X 0,Y 341.026,Z 232.006,A -85,B 0,C 180,E1 -14302.897,E2 -14302.897} C_VEL
LIN {X 0,Y 341.118,Z 231.992,A -85,B 0,C 180,E1 -14307.638,E2 -14307.638} C_VEL
LIN {X 0,Y 341.257,Z 231.973,A -85,B 0,C 180,E1 -14310,E2 -14310} C_VEL
LIN {X 0,Y 341.118,Z 231.991,A -85,B 0,C 180,E1 -14312.361,E2 -14312.361} C_VEL
LIN {X 0,Y 341.018,Z 232.009,A -85,B 0,C 180,E1 -14317.103,E2 -14317.103} C_VEL
LIN {X 0,Y 340.996,Z 232.189,A -85,B 0,C 180,E1 -14317.896,E2 -14317.896} C_VEL
LIN {X 0,Y 342.324,Z 239.627,A -85,B 0,C 180,E1 -14320.051,E2 -14320.051} C_VEL
LIN {X 0,Y 347.225,Z 253.856,A -85,B 0,C 180,E1 -14320.686,E2 -14320.686} C_VEL
LIN {X 0,Y 349.652,Z 266.246,A -85,B 0,C 180,E1 -14321.117,E2 -14321.117} C_VEL
LIN {X 0,Y 347.943,Z 347.643,A -85,B 0,C 180,E1 -14322.894,E2 -14322.894} C_VEL
LIN {X 0,Y 347.324,Z 360.647,A -85,B 0,C 180,E1 -14323.407,E2 -14323.407} C_VEL
LIN {X 0,Y 346.65,Z 373.401,A -85,B 0,C 180,E1 -14324.155,E2 -14324.155} C_VEL
LIN {X 0,Y 345.807,Z 384.383,A -85,B 0,C 180,E1 -14325.018,E2 -14325.018} C_VEL
LIN {X 0,Y 344.823,Z 395.41,A -85,B 0,C 180,E1 -14326.122,E2 -14326.122} C_VEL
LIN {X 0,Y 343.762,Z 405.629,A -85,B 0,C 180,E1 -14327.397,E2 -14327.397} C_VEL
LIN {X 0,Y 342.626,Z 415.083,A -85,B 0,C 180,E1 -14328.848,E2 -14328.848} C_VEL
LIN {X 0,Y 341.689,Z 423.552,A -85,B 0,C 180,E1 -14330.466,E2 -14330.466} C_VEL
LIN {X 0,Y 340.957,Z 430.02,A -85,B 0,C 180,E1 -14331.968,E2 -14331.968} C_VEL
LIN {X 0,Y 340.31,Z 436.236,A -85,B 0,C 180,E1 -14333.747,E2 -14333.747} C_VEL
LIN {X 0,Y 339.734,Z 441.705,A -85,B 0,C 180,E1 -14335.748,E2 -14335.748} C_VEL
LIN {X 0,Y 339.452,Z 445.793,A -85,B 0,C 180,E1 -14337.763,E2 -14337.763} C_VEL
LIN {X 0,Y 339.028,Z 448.634,A -85,B 0,C 180,E1 -14339.835,E2 -14339.835} C_VEL
LIN {X 0,Y 338.869,Z 450.142,A -85,B 0,C 180,E1 -14341.771,E2 -14341.771} C_VEL
LIN {X 0,Y 338.873,Z 450.544,A -85,B 0,C 180,E1 -14344.052,E2 -14344.052} C_VEL
LIN {X 0,Y 339.029,Z 449.686,A -85,B 0,C 180,E1 -14346.07,E2 -14346.07} C_VEL
LIN {X 0,Y 339.363,Z 447.364,A -85,B 0,C 180,E1 -14348.308,E2 -14348.308} C_VEL
LIN {X 0,Y 338.906,Z 445.957,A -85,B 0,C 180,E1 -14349.274,E2 -14349.274} C_VEL
LIN {X 0,Y 336.479,Z 443.291,A -85,B 0,C 180,E1 -14350.843,E2 -14350.843} C_VEL
LIN {X 0,Y 334.489,Z 440.682,A -85,B 0,C 180,E1 -14352.082,E2 -14352.082} C_VEL
LIN {X 0,Y 333.813,Z 438.343,A -85,B 0,C 180,E1 -14353.008,E2 -14353.008} C_VEL
LIN {X 0,Y 333.857,Z 437.457,A -85,B 0,C 180,E1 -14353.313,E2 -14353.313} C_VEL
LIN {X 0,Y 334.793,Z 431.204,A -85,B 0,C 180,E1 -14355.202,E2 -14355.202} C_VEL
LIN {X 0,Y 335.973,Z 423.444,A -85,B 0,C 180,E1 -14357.065,E2 -14357.065} C_VEL
LIN {X 0,Y 337.373,Z 414.223,A -85,B 0,C 180,E1 -14358.809,E2 -14358.809} C_VEL
LIN {X 0,Y 338.829,Z 404.02,A -85,B 0,C 180,E1 -14360.356,E2 -14360.356} C_VEL
LIN {X 0,Y 340.097,Z 393.814,A -85,B 0,C 180,E1 -14361.596,E2 -14361.596} C_VEL
LIN {X 0,Y 341.331,Z 382.524,A -85,B 0,C 180,E1 -14362.68,E2 -14362.68} C_VEL
LIN {X 0,Y 342.416,Z 370.322,A -85,B 0,C 180,E1 -14363.584,E2 -14363.584} C_VEL
LIN {X 0,Y 343.23,Z 357.652,A -85,B 0,C 180,E1 -14364.266,E2 -14364.266} C_VEL
LIN {X 0,Y 343.814,Z 344.125,A -85,B 0,C 180,E1 -14364.728,E2 -14364.728} C_VEL
LIN {X 0,Y 345.754,Z 268.388,A -85,B 0,C 180,E1 -14366.419,E2 -14366.419} C_VEL
LIN {X 0,Y 343.643,Z 259.417,A -85,B 0,C 180,E1 -14366.819,E2 -14366.819} C_VEL
LIN {X 0,Y 336.663,Z 243.214,A -85,B 0,C 180,E1 -14367.847,E2 -14367.847} C_VEL
LIN {X 0,Y 335.42,Z 240.322,A -85,B 0,C 180,E1 -14368.068,E2 -14368.068} C_VEL
LIN {X 0,Y 333.716,Z 232.919,A -85,B 0,C 180,E1 -14370.346,E2 -14370.346} C_VEL
LIN {X 0,Y 333.707,Z 232.915,A -85,B 0,C 180,E1 -14373.761,E2 -14373.761} C_VEL
LIN {X 0,Y 333.694,Z 232.917,A -85,B 0,C 180,E1 -14377.921,E2 -14377.921} C_VEL
LIN {X 0,Y 333.771,Z 232.912,A -85,B 0,C 180,E1 -14381.596,E2 -14381.596} C_VEL
LIN {X 0,Y 333.789,Z 232.904,A -85,B 0,C 180,E1 -14385.584,E2 -14385.584} C_VEL
LIN {X 0,Y 333.819,Z 232.903,A -85,B 0,C 180,E1 -14389.085,E2 -14389.085} C_VEL
LIN {X 0,Y 333.975,Z 232.884,A -85,B 0,C 180,E1 -14392.754,E2 -14392.754} C_VEL
LIN {X 0,Y 333.787,Z 232.903,A -85,B 0,C 180,E1 -14395.176,E2 -14395.176} C_VEL
LIN {X 0,Y 334.091,Z 232.865,A -85,B 0,C 180,E1 -14397.596,E2 -14397.596} C_VEL
LIN {X 0,Y 334.197,Z 232.854,A -85,B 0,C 180,E1 -14400.007,E2 -14400.007} C_VEL
LIN {X 0,Y 334.06,Z 232.865,A -85,B 0,C 180,E1 -14402.418,E2 -14402.418} C_VEL
LIN {X 0,Y 333.995,Z 232.872,A -85,B 0,C 180,E1 -14406.046,E2 -14406.046} C_VEL
LIN {X 0,Y 333.816,Z 232.895,A -85,B 0,C 180,E1 -14409.703,E2 -14409.703} C_VEL
LIN {X 0,Y 333.791,Z 232.901,A -85,B 0,C 180,E1 -14413.398,E2 -14413.398} C_VEL
LIN {X 0,Y 333.719,Z 232.912,A -85,B 0,C 180,E1 -14417.154,E2 -14417.154} C_VEL
LIN {X 0,Y 333.666,Z 232.918,A -85,B 0,C 180,E1 -14419.701,E2 -14419.701} C_VEL
LIN {X 0,Y 333.645,Z 232.92,A -85,B 0,C 180,E1 -14423.598,E2 -14423.598} C_VEL
LIN {X 0,Y 333.632,Z 232.92,A -85,B 0,C 180,E1 -14426.261,E2 -14426.261} C_VEL
LIN {X 0,Y 333.634,Z 232.923,A -85,B 0,C 180,E1 -14428.985,E2 -14428.985} C_VEL
LIN {X 0,Y 333.645,Z 232.922,A -85,B 0,C 180,E1 -14432.59,E2 -14432.59} C_VEL
LIN {X 0,Y 333.681,Z 232.919,A -85,B 0,C 180,E1 -14436.144,E2 -14436.144} C_VEL
LIN {X 0,Y 333.611,Z 232.926,A -85,B 0,C 180,E1 -14439.203,E2 -14439.203} C_VEL
LIN {X 0,Y 333.617,Z 232.929,A -85,B 0,C 180,E1 -14442.499,E2 -14442.499} C_VEL
LIN {X 0,Y 333.594,Z 232.936,A -85,B 0,C 180,E1 -14445.956,E2 -14445.956} C_VEL
LIN {X 0,Y 333.61,Z 232.93,A -85,B 0,C 180,E1 -14449.329,E2 -14449.329} C_VEL
LIN {X 0,Y 333.673,Z 232.922,A -85,B 0,C 180,E1 -14453.173,E2 -14453.173} C_VEL
LIN {X 0,Y 333.686,Z 232.921,A -85,B 0,C 180,E1 -14455.344,E2 -14455.344} C_VEL
LIN {X 0,Y 333.652,Z 232.982,A -85,B 0,C 180,E1 -14457.418,E2 -14457.418} C_VEL
LIN {X 0,Y 335.973,Z 242.458,A -85,B 0,C 180,E1 -14460.212,E2 -14460.212} C_VEL
LIN {X 0,Y 338.259,Z 253.634,A -85,B 0,C 180,E1 -14463.313,E2 -14463.313} C_VEL
LIN {X 0,Y 338.582,Z 256.88,A -85,B 0,C 180,E1 -14464.158,E2 -14464.158} C_VEL
LIN {X 0,Y 338.125,Z 261.402,A -85,B 0,C 180,E1 -14465.251,E2 -14465.251} C_VEL
LIN {X 0,Y 342.9,Z 286.455,A -85,B 0,C 180,E1 -14466.293,E2 -14466.293} C_VEL
LIN {X 0,Y 345.049,Z 301.595,A -85,B 0,C 180,E1 -14466.841,E2 -14466.841} C_VEL
LIN {X 0,Y 343.334,Z 371.236,A -85,B 0,C 180,E1 -14468.42,E2 -14468.42} C_VEL
LIN {X 0,Y 342.395,Z 384.72,A -85,B 0,C 180,E1 -14468.949,E2 -14468.949} C_VEL
LIN {X 0,Y 341.31,Z 397.015,A -85,B 0,C 180,E1 -14469.668,E2 -14469.668} C_VEL
LIN {X 0,Y 340.141,Z 408.08,A -85,B 0,C 180,E1 -14470.539,E2 -14470.539} C_VEL
LIN {X 0,Y 338.622,Z 419.655,A -85,B 0,C 180,E1 -14471.705,E2 -14471.705} C_VEL
LIN {X 0,Y 337.239,Z 430.111,A -85,B 0,C 180,E1 -14473.037,E2 -14473.037} C_VEL
LIN {X 0,Y 335.966,Z 439.552,A -85,B 0,C 180,E1 -14474.532,E2 -14474.532} C_VEL
LIN {X 0,Y 334.676,Z 448.689,A -85,B 0,C 180,E1 -14476.336,E2 -14476.336} C_VEL
LIN {X 0,Y 333.517,Z 456.075,A -85,B 0,C 180,E1 -14478.144,E2 -14478.144} C_VEL
LIN {X 0,Y 332.927,Z 461.094,A -85,B 0,C 180,E1 -14479.664,E2 -14479.664} C_VEL
LIN {X 0,Y 332.432,Z 465.988,A -85,B 0,C 180,E1 -14481.49,E2 -14481.49} C_VEL
LIN {X 0,Y 332.093,Z 469.76,A -85,B 0,C 180,E1 -14483.316,E2 -14483.316} C_VEL
LIN {X 0,Y 331.963,Z 472.51,A -85,B 0,C 180,E1 -14485.142,E2 -14485.142} C_VEL
LIN {X 0,Y 331.998,Z 473.819,A -85,B 0,C 180,E1 -14486.359,E2 -14486.359} C_VEL
LIN {X 0,Y 331.948,Z 474.718,A -85,B 0,C 180,E1 -14487.573,E2 -14487.573} C_VEL
LIN {X 0,Y 331.962,Z 475.175,A -85,B 0,C 180,E1 -14488.787,E2 -14488.787} C_VEL
LIN {X 0,Y 332.023,Z 475.236,A -85,B 0,C 180,E1 -14490,E2 -14490} C_VEL
LIN {X 0,Y 331.977,Z 474.9,A -85,B 0,C 180,E1 -14491.213,E2 -14491.213} C_VEL
LIN {X 0,Y 331.952,Z 474.162,A -85,B 0,C 180,E1 -14492.427,E2 -14492.427} C_VEL
LIN {X 0,Y 332.008,Z 472.972,A -85,B 0,C 180,E1 -14493.641,E2 -14493.641} C_VEL
LIN {X 0,Y 332.044,Z 469.787,A -85,B 0,C 180,E1 -14495.814,E2 -14495.814} C_VEL
LIN {X 0,Y 332.289,Z 465.355,A -85,B 0,C 180,E1 -14497.902,E2 -14497.902} C_VEL
LIN {X 0,Y 332.768,Z 459.221,A -85,B 0,C 180,E1 -14500.034,E2 -14500.034} C_VEL
LIN {X 0,Y 333.4,Z 452.487,A -85,B 0,C 180,E1 -14501.86,E2 -14501.86} C_VEL
LIN {X 0,Y 334.432,Z 444.13,A -85,B 0,C 180,E1 -14503.675,E2 -14503.675} C_VEL
LIN {X 0,Y 335.554,Z 434.387,A -85,B 0,C 180,E1 -14505.358,E2 -14505.358} C_VEL
LIN {X 0,Y 336.649,Z 423.715,A -85,B 0,C 180,E1 -14506.837,E2 -14506.837} C_VEL
LIN {X 0,Y 337.827,Z 412.922,A -85,B 0,C 180,E1 -14508.026,E2 -14508.026} C_VEL
LIN {X 0,Y 338.996,Z 400.823,A -85,B 0,C 180,E1 -14509.058,E2 -14509.058} C_VEL
LIN {X 0,Y 340.078,Z 388.262,A -85,B 0,C 180,E1 -14509.858,E2 -14509.858} C_VEL
LIN {X 0,Y 340.757,Z 376.132,A -85,B 0,C 180,E1 -14510.406,E2 -14510.406} C_VEL
LIN {X 0,Y 341.25,Z 360.259,A -85,B 0,C 180,E1 -14510.829,E2 -14510.829} C_VEL
LIN {X 0,Y 342.419,Z 299.996,A -85,B 0,C 180,E1 -14512.153,E2 -14512.153} C_VEL
LIN {X 0,Y 336.844,Z 262.892,A -85,B 0,C 180,E1 -14513.384,E2 -14513.384} C_VEL
LIN {X 0,Y 337.77,Z 253.899,A -85,B 0,C 180,E1 -14515.578,E2 -14515.578} C_VEL
LIN {X 0,Y 336.165,Z 244.811,A -85,B 0,C 180,E1 -14517.994,E2 -14517.994} C_VEL
LIN {X 0,Y 333.67,Z 232.921,A -85,B 0,C 180,E1 -14521.308,E2 -14521.308} C_VEL
LIN {X 0,Y 333.682,Z 232.917,A -85,B 0,C 180,E1 -14524.766,E2 -14524.766} C_VEL
LIN {X 0,Y 333.653,Z 232.925,A -85,B 0,C 180,E1 -14527.65,E2 -14527.65} C_VEL
LIN {X 0,Y 333.605,Z 232.927,A -85,B 0,C 180,E1 -14530.772,E2 -14530.772} C_VEL
LIN {X 0,Y 333.576,Z 232.932,A -85,B 0,C 180,E1 -14534.241,E2 -14534.241} C_VEL
LIN {X 0,Y 333.623,Z 232.929,A -85,B 0,C 180,E1 -14537.609,E2 -14537.609} C_VEL
LIN {X 0,Y 333.624,Z 232.926,A -85,B 0,C 180,E1 -14541.207,E2 -14541.207} C_VEL
LIN {X 0,Y 333.679,Z 232.922,A -85,B 0,C 180,E1 -14543.855,E2 -14543.855} C_VEL
LIN {X 0,Y 333.645,Z 232.925,A -85,B 0,C 180,E1 -14547.41,E2 -14547.41} C_VEL
LIN {X 0,Y 333.629,Z 232.924,A -85,B 0,C 180,E1 -14551.014,E2 -14551.014} C_VEL
LIN {X 0,Y 333.663,Z 232.919,A -85,B 0,C 180,E1 -14554.917,E2 -14554.917} C_VEL
LIN {X 0,Y 333.653,Z 232.921,A -85,B 0,C 180,E1 -14559.011,E2 -14559.011} C_VEL
LIN {X 0,Y 333.698,Z 232.914,A -85,B 0,C 180,E1 -14562.845,E2 -14562.845} C_VEL
LIN {X 0,Y 333.808,Z 232.907,A -85,B 0,C 180,E1 -14565.571,E2 -14565.571} C_VEL
LIN {X 0,Y 333.805,Z 232.903,A -85,B 0,C 180,E1 -14569.071,E2 -14569.071} C_VEL
LIN {X 0,Y 333.95,Z 232.883,A -85,B 0,C 180,E1 -14572.739,E2 -14572.739} C_VEL
LIN {X 0,Y 333.763,Z 232.908,A -85,B 0,C 180,E1 -14575.162,E2 -14575.162} C_VEL
LIN {X 0,Y 334.028,Z 232.878,A -85,B 0,C 180,E1 -14577.582,E2 -14577.582} C_VEL
LIN {X 0,Y 334.047,Z 232.874,A -85,B 0,C 180,E1 -14581.199,E2 -14581.199} C_VEL
LIN {X 0,Y 334.057,Z 232.87,A -85,B 0,C 180,E1 -14582.405,E2 -14582.405} C_VEL
LIN {X 0,Y 333.94,Z 232.884,A -85,B 0,C 180,E1 -14586.485,E2 -14586.485} C_VEL
LIN {X 0,Y 333.802,Z 232.905,A -85,B 0,C 180,E1 -14589.689,E2 -14589.689} C_VEL
LIN {X 0,Y 333.773,Z 232.911,A -85,B 0,C 180,E1 -14593.385,E2 -14593.385} C_VEL
LIN {X 0,Y 333.736,Z 232.912,A -85,B 0,C 180,E1 -14595.88,E2 -14595.88} C_VEL
LIN {X 0,Y 333.698,Z 232.918,A -85,B 0,C 180,E1 -14599.684,E2 -14599.684} C_VEL
LIN {X 0,Y 333.642,Z 232.926,A -85,B 0,C 180,E1 -14603.583,E2 -14603.583} C_VEL
LIN {X 0,Y 333.662,Z 232.919,A -85,B 0,C 180,E1 -14606.243,E2 -14606.243} C_VEL
LIN {X 0,Y 333.653,Z 232.922,A -85,B 0,C 180,E1 -14608.968,E2 -14608.968} C_VEL
LIN {X 0,Y 333.603,Z 232.93,A -85,B 0,C 180,E1 -14613.202,E2 -14613.202} C_VEL
LIN {X 0,Y 333.639,Z 232.922,A -85,B 0,C 180,E1 -14616.133,E2 -14616.133} C_VEL
LIN {X 0,Y 333.608,Z 232.931,A -85,B 0,C 180,E1 -14619.186,E2 -14619.186} C_VEL
LIN {X 0,Y 333.591,Z 232.928,A -85,B 0,C 180,E1 -14622.494,E2 -14622.494} C_VEL
LIN {X 0,Y 333.578,Z 232.93,A -85,B 0,C 180,E1 -14625.953,E2 -14625.953} C_VEL
LIN {X 0,Y 333.601,Z 232.932,A -85,B 0,C 180,E1 -14629.31,E2 -14629.31} C_VEL
LIN {X 0,Y 333.616,Z 232.93,A -85,B 0,C 180,E1 -14633.163,E2 -14633.163} C_VEL
LIN {X 0,Y 333.624,Z 232.929,A -85,B 0,C 180,E1 -14635.336,E2 -14635.336} C_VEL
LIN {X 0,Y 333.651,Z 232.922,A -85,B 0,C 180,E1 -14639.706,E2 -14639.706} C_VEL
LIN {X 0,Y 333.691,Z 232.916,A -85,B 0,C 180,E1 -14642.397,E2 -14642.397} C_VEL
LIN {X 0,Y 333.706,Z 232.919,A -85,B 0,C 180,E1 -14645.09,E2 -14645.09} C_VEL
LIN {X 0,Y 333.665,Z 232.924,A -85,B 0,C 180,E1 -14649.019,E2 -14649.019} C_VEL
LIN {X 0,Y 333.739,Z 232.912,A -85,B 0,C 180,E1 -14651.587,E2 -14651.587} C_VEL
LIN {X 0,Y 333.751,Z 232.91,A -85,B 0,C 180,E1 -14655.575,E2 -14655.575} C_VEL
LIN {X 0,Y 333.779,Z 232.911,A -85,B 0,C 180,E1 -14659.076,E2 -14659.076} C_VEL
LIN {X 0,Y 333.974,Z 232.883,A -85,B 0,C 180,E1 -14662.747,E2 -14662.747} C_VEL
LIN {X 0,Y 333.763,Z 232.912,A -85,B 0,C 180,E1 -14665.168,E2 -14665.168} C_VEL
LIN {X 0,Y 334.079,Z 232.869,A -85,B 0,C 180,E1 -14667.589,E2 -14667.589} C_VEL
LIN {X 0,Y 334.207,Z 232.851,A -85,B 0,C 180,E1 -14670,E2 -14670} C_VEL
LIN {X 0,Y 334.08,Z 232.868,A -85,B 0,C 180,E1 -14672.411,E2 -14672.411} C_VEL
LIN {X 0,Y 333.968,Z 232.887,A -85,B 0,C 180,E1 -14677.253,E2 -14677.253} C_VEL
LIN {X 0,Y 333.958,Z 233.004,A -85,B 0,C 180,E1 -14677.558,E2 -14677.558} C_VEL
LIN {X 0,Y 335.176,Z 239.977,A -85,B 0,C 180,E1 -14679.596,E2 -14679.596} C_VEL
LIN {X 0,Y 340.747,Z 255.832,A -85,B 0,C 180,E1 -14680.33,E2 -14680.33} C_VEL
LIN {X 0,Y 343.049,Z 267.768,A -85,B 0,C 180,E1 -14680.753,E2 -14680.753} C_VEL
LIN {X 0,Y 341.201,Z 347.753,A -85,B 0,C 180,E1 -14682.528,E2 -14682.528} C_VEL
LIN {X 0,Y 340.56,Z 361.429,A -85,B 0,C 180,E1 -14683.082,E2 -14683.082} C_VEL
LIN {X 0,Y 339.818,Z 374.168,A -85,B 0,C 180,E1 -14683.855,E2 -14683.855} C_VEL
LIN {X 0,Y 338.873,Z 386.471,A -85,B 0,C 180,E1 -14684.871,E2 -14684.871} C_VEL
LIN {X 0,Y 337.731,Z 397.949,A -85,B 0,C 180,E1 -14686.085,E2 -14686.085} C_VEL
LIN {X 0,Y 336.587,Z 408.258,A -85,B 0,C 180,E1 -14687.466,E2 -14687.466} C_VEL
LIN {X 0,Y 335.476,Z 417.143,A -85,B 0,C 180,E1 -14688.93,E2 -14688.93} C_VEL
LIN {X 0,Y 334.552,Z 425.383,A -85,B 0,C 180,E1 -14690.601,E2 -14690.601} C_VEL
LIN {X 0,Y 333.775,Z 432.086,A -85,B 0,C 180,E1 -14692.272,E2 -14692.272} C_VEL
LIN {X 0,Y 333.051,Z 438.322,A -85,B 0,C 180,E1 -14694.214,E2 -14694.214} C_VEL
LIN {X 0,Y 332.537,Z 443.507,A -85,B 0,C 180,E1 -14696.347,E2 -14696.347} C_VEL
LIN {X 0,Y 332.212,Z 447.158,A -85,B 0,C 180,E1 -14698.423,E2 -14698.423} C_VEL
LIN {X 0,Y 331.837,Z 449.595,A -85,B 0,C 180,E1 -14700.55,E2 -14700.55} C_VEL
LIN {X 0,Y 331.758,Z 450.531,A -85,B 0,C 180,E1 -14702.092,E2 -14702.092} C_VEL
LIN {X 0,Y 331.783,Z 450.789,A -85,B 0,C 180,E1 -14704.315,E2 -14704.315} C_VEL
LIN {X 0,Y 331.981,Z 449.767,A -85,B 0,C 180,E1 -14706.458,E2 -14706.458} C_VEL
LIN {X 0,Y 332.329,Z 447.55,A -85,B 0,C 180,E1 -14708.528,E2 -14708.528} C_VEL
LIN {X 0,Y 332.941,Z 443.538,A -85,B 0,C 180,E1 -14710.871,E2 -14710.871} C_VEL
LIN {X 0,Y 333.801,Z 437.861,A -85,B 0,C 180,E1 -14713.176,E2 -14713.176} C_VEL
LIN {X 0,Y 333.857,Z 437.457,A -85,B 0,C 180,E1 -14713.313,E2 -14713.313} C_VEL
LIN {X 0,Y 333.596,Z 434.784,A -85,B 0,C 180,E1 -14714.216,E2 -14714.216} C_VEL
LIN {X 0,Y 331.505,Z 430.145,A -85,B 0,C 180,E1 -14715.687,E2 -14715.687} C_VEL
LIN {X 0,Y 329.576,Z 424.934,A -85,B 0,C 180,E1 -14717.108,E2 -14717.108} C_VEL
LIN {X 0,Y 329.557,Z 421.297,A -85,B 0,C 180,E1 -14717.918,E2 -14717.918} C_VEL
LIN {X 0,Y 330.902,Z 412.634,A -85,B 0,C 180,E1 -14719.515,E2 -14719.515} C_VEL
LIN {X 0,Y 332.315,Z 403.166,A -85,B 0,C 180,E1 -14720.923,E2 -14720.923} C_VEL
LIN {X 0,Y 333.74,Z 391.909,A -85,B 0,C 180,E1 -14722.267,E2 -14722.267} C_VEL
LIN {X 0,Y 335.039,Z 380.314,A -85,B 0,C 180,E1 -14723.354,E2 -14723.354} C_VEL
LIN {X 0,Y 336.098,Z 368.041,A -85,B 0,C 180,E1 -14724.223,E2 -14724.223} C_VEL
LIN {X 0,Y 336.975,Z 354.26,A -85,B 0,C 180,E1 -14724.91,E2 -14724.91} C_VEL
LIN {X 0,Y 337.533,Z 340.193,A -85,B 0,C 180,E1 -14725.329,E2 -14725.329} C_VEL
LIN {X 0,Y 339.356,Z 269.158,A -85,B 0,C 180,E1 -14726.946,E2 -14726.946} C_VEL
LIN {X 0,Y 337.582,Z 261.97,A -85,B 0,C 180,E1 -14727.283,E2 -14727.283} C_VEL
LIN {X 0,Y 330.8,Z 246.282,A -85,B 0,C 180,E1 -14728.322,E2 -14728.322} C_VEL
LIN {X 0,Y 328.306,Z 240.685,A -85,B 0,C 180,E1 -14728.738,E2 -14728.738} C_VEL
LIN {X 0,Y 326.651,Z 233.797,A -85,B 0,C 180,E1 -14730.969,E2 -14730.969} C_VEL
LIN {X 0,Y 326.66,Z 233.796,A -85,B 0,C 180,E1 -14734.634,E2 -14734.634} C_VEL
LIN {X 0,Y 326.621,Z 233.801,A -85,B 0,C 180,E1 -14738.552,E2 -14738.552} C_VEL
LIN {X 0,Y 326.722,Z 233.792,A -85,B 0,C 180,E1 -14741.185,E2 -14741.185} C_VEL
LIN {X 0,Y 326.744,Z 233.782,A -85,B 0,C 180,E1 -14745.441,E2 -14745.441} C_VEL
LIN {X 0,Y 326.755,Z 233.781,A -85,B 0,C 180,E1 -14748.846,E2 -14748.846} C_VEL
LIN {X 0,Y 326.925,Z 233.76,A -85,B 0,C 180,E1 -14752.597,E2 -14752.597} C_VEL
LIN {X 0,Y 326.754,Z 233.779,A -85,B 0,C 180,E1 -14755.072,E2 -14755.072} C_VEL
LIN {X 0,Y 327.032,Z 233.744,A -85,B 0,C 180,E1 -14757.544,E2 -14757.544} C_VEL
LIN {X 0,Y 327.149,Z 233.732,A -85,B 0,C 180,E1 -14760.007,E2 -14760.007} C_VEL
LIN {X 0,Y 327.003,Z 233.744,A -85,B 0,C 180,E1 -14762.47,E2 -14762.47} C_VEL
LIN {X 0,Y 326.951,Z 233.749,A -85,B 0,C 180,E1 -14766.177,E2 -14766.177} C_VEL
LIN {X 0,Y 326.779,Z 233.771,A -85,B 0,C 180,E1 -14769.914,E2 -14769.914} C_VEL
LIN {X 0,Y 326.755,Z 233.777,A -85,B 0,C 180,E1 -14773.692,E2 -14773.692} C_VEL
LIN {X 0,Y 326.665,Z 233.79,A -85,B 0,C 180,E1 -14777.536,E2 -14777.536} C_VEL
LIN {X 0,Y 326.614,Z 233.796,A -85,B 0,C 180,E1 -14781.463,E2 -14781.463} C_VEL
LIN {X 0,Y 326.605,Z 233.797,A -85,B 0,C 180,E1 -14785.497,E2 -14785.497} C_VEL
LIN {X 0,Y 326.595,Z 233.803,A -85,B 0,C 180,E1 -14788.262,E2 -14788.262} C_VEL
LIN {X 0,Y 326.574,Z 233.804,A -85,B 0,C 180,E1 -14791.103,E2 -14791.103} C_VEL
LIN {X 0,Y 326.613,Z 233.794,A -85,B 0,C 180,E1 -14794.025,E2 -14794.025} C_VEL
LIN {X 0,Y 326.63,Z 233.796,A -85,B 0,C 180,E1 -14797.241,E2 -14797.241} C_VEL
LIN {X 0,Y 326.544,Z 233.811,A -85,B 0,C 180,E1 -14801.126,E2 -14801.126} C_VEL
LIN {X 0,Y 326.527,Z 233.813,A -85,B 0,C 180,E1 -14804.744,E2 -14804.744} C_VEL
LIN {X 0,Y 326.559,Z 233.813,A -85,B 0,C 180,E1 -14808.153,E2 -14808.153} C_VEL
LIN {X 0,Y 326.579,Z 233.805,A -85,B 0,C 180,E1 -14811.386,E2 -14811.386} C_VEL
LIN {X 0,Y 326.631,Z 233.801,A -85,B 0,C 180,E1 -14814.856,E2 -14814.856} C_VEL
LIN {X 0,Y 326.635,Z 233.982,A -85,B 0,C 180,E1 -14816.879,E2 -14816.879} C_VEL
LIN {X 0,Y 329.068,Z 243.84,A -85,B 0,C 180,E1 -14819.875,E2 -14819.875} C_VEL
LIN {X 0,Y 331.326,Z 254.789,A -85,B 0,C 180,E1 -14822.994,E2 -14822.994} C_VEL
LIN {X 0,Y 331.753,Z 258.238,A -85,B 0,C 180,E1 -14823.924,E2 -14823.924} C_VEL
LIN {X 0,Y 331.484,Z 261.028,A -85,B 0,C 180,E1 -14824.618,E2 -14824.618} C_VEL
LIN {X 0,Y 336.357,Z 286.36,A -85,B 0,C 180,E1 -14825.731,E2 -14825.731} C_VEL
LIN {X 0,Y 338.671,Z 303.115,A -85,B 0,C 180,E1 -14826.351,E2 -14826.351} C_VEL
LIN {X 0,Y 336.864,Z 370.721,A -85,B 0,C 180,E1 -14827.912,E2 -14827.912} C_VEL
LIN {X 0,Y 335.858,Z 384.823,A -85,B 0,C 180,E1 -14828.479,E2 -14828.479} C_VEL
LIN {X 0,Y 334.7,Z 397.474,A -85,B 0,C 180,E1 -14829.248,E2 -14829.248} C_VEL
LIN {X 0,Y 333.481,Z 408.354,A -85,B 0,C 180,E1 -14830.134,E2 -14830.134} C_VEL
LIN {X 0,Y 331.907,Z 419.832,A -85,B 0,C 180,E1 -14831.322,E2 -14831.322} C_VEL
LIN {X 0,Y 330.445,Z 430.213,A -85,B 0,C 180,E1 -14832.678,E2 -14832.678} C_VEL
LIN {X 0,Y 329.112,Z 439.619,A -85,B 0,C 180,E1 -14834.211,E2 -14834.211} C_VEL
LIN {X 0,Y 327.773,Z 448.66,A -85,B 0,C 180,E1 -14836.042,E2 -14836.042} C_VEL
LIN {X 0,Y 326.556,Z 456.007,A -85,B 0,C 180,E1 -14837.888,E2 -14837.888} C_VEL
LIN {X 0,Y 325.913,Z 460.989,A -85,B 0,C 180,E1 -14839.439,E2 -14839.439} C_VEL
LIN {X 0,Y 325.378,Z 465.847,A -85,B 0,C 180,E1 -14841.304,E2 -14841.304} C_VEL
LIN {X 0,Y 325.016,Z 469.584,A -85,B 0,C 180,E1 -14843.17,E2 -14843.17} C_VEL
LIN {X 0,Y 324.876,Z 472.304,A -85,B 0,C 180,E1 -14845.036,E2 -14845.036} C_VEL
LIN {X 0,Y 324.901,Z 473.599,A -85,B 0,C 180,E1 -14846.279,E2 -14846.279} C_VEL
LIN {X 0,Y 324.866,Z 474.477,A -85,B 0,C 180,E1 -14847.52,E2 -14847.52} C_VEL
LIN {X 0,Y 324.87,Z 474.917,A -85,B 0,C 180,E1 -14848.761,E2 -14848.761} C_VEL
LIN {X 0,Y 324.928,Z 474.966,A -85,B 0,C 180,E1 -14850,E2 -14850} C_VEL
LIN {X 0,Y 324.883,Z 474.618,A -85,B 0,C 180,E1 -14851.24,E2 -14851.24} C_VEL
LIN {X 0,Y 324.87,Z 473.859,A -85,B 0,C 180,E1 -14852.48,E2 -14852.48} C_VEL
LIN {X 0,Y 324.912,Z 472.65,A -85,B 0,C 180,E1 -14853.721,E2 -14853.721} C_VEL
LIN {X 0,Y 324.94,Z 469.778,A -85,B 0,C 180,E1 -14855.743,E2 -14855.743} C_VEL
LIN {X 0,Y 325.222,Z 464.971,A -85,B 0,C 180,E1 -14858.075,E2 -14858.075} C_VEL
LIN {X 0,Y 325.725,Z 458.784,A -85,B 0,C 180,E1 -14860.253,E2 -14860.253} C_VEL
LIN {X 0,Y 326.431,Z 452.012,A -85,B 0,C 180,E1 -14862.117,E2 -14862.117} C_VEL
LIN {X 0,Y 327.459,Z 443.601,A -85,B 0,C 180,E1 -14863.972,E2 -14863.972} C_VEL
LIN {X 0,Y 328.546,Z 434.765,A -85,B 0,C 180,E1 -14865.535,E2 -14865.535} C_VEL
LIN {X 0,Y 329.676,Z 424.221,A -85,B 0,C 180,E1 -14867.045,E2 -14867.045} C_VEL
LIN {X 0,Y 330.885,Z 413.611,A -85,B 0,C 180,E1 -14868.257,E2 -14868.257} C_VEL
LIN {X 0,Y 332.083,Z 401.837,A -85,B 0,C 180,E1 -14869.309,E2 -14869.309} C_VEL
LIN {X 0,Y 333.108,Z 389.641,A -85,B 0,C 180,E1 -14870.13,E2 -14870.13} C_VEL
LIN {X 0,Y 333.989,Z 376.424,A -85,B 0,C 180,E1 -14870.758,E2 -14870.758} C_VEL
LIN {X 0,Y 334.489,Z 361.572,A -85,B 0,C 180,E1 -14871.176,E2 -14871.176} C_VEL
LIN {X 0,Y 335.753,Z 301.124,A -85,B 0,C 180,E1 -14872.529,E2 -14872.529} C_VEL
LIN {X 0,Y 330.023,Z 262.68,A -85,B 0,C 180,E1 -14873.824,E2 -14873.824} C_VEL
LIN {X 0,Y 330.78,Z 254.689,A -85,B 0,C 180,E1 -14875.82,E2 -14875.82} C_VEL
LIN {X 0,Y 328.768,Z 243.896,A -85,B 0,C 180,E1 -14878.775,E2 -14878.775} C_VEL
LIN {X 0,Y 326.603,Z 233.805,A -85,B 0,C 180,E1 -14881.68,E2 -14881.68} C_VEL
LIN {X 0,Y 326.616,Z 233.801,A -85,B 0,C 180,E1 -14885.518,E2 -14885.518} C_VEL
LIN {X 0,Y 326.578,Z 233.802,A -85,B 0,C 180,E1 -14888.614,E2 -14888.614} C_VEL
LIN {X 0,Y 326.541,Z 233.812,A -85,B 0,C 180,E1 -14891.85,E2 -14891.85} C_VEL
LIN {X 0,Y 326.522,Z 233.811,A -85,B 0,C 180,E1 -14895.257,E2 -14895.257} C_VEL
LIN {X 0,Y 326.543,Z 233.806,A -85,B 0,C 180,E1 -14898.874,E2 -14898.874} C_VEL
LIN {X 0,Y 326.628,Z 233.796,A -85,B 0,C 180,E1 -14902.76,E2 -14902.76} C_VEL
LIN {X 0,Y 326.613,Z 233.801,A -85,B 0,C 180,E1 -14905.975,E2 -14905.975} C_VEL
LIN {X 0,Y 326.611,Z 233.801,A -85,B 0,C 180,E1 -14909.395,E2 -14909.395} C_VEL
LIN {X 0,Y 326.601,Z 233.8,A -85,B 0,C 180,E1 -14913.129,E2 -14913.129} C_VEL
LIN {X 0,Y 326.616,Z 233.801,A -85,B 0,C 180,E1 -14915.862,E2 -14915.862} C_VEL
LIN {X 0,Y 326.611,Z 233.797,A -85,B 0,C 180,E1 -14918.537,E2 -14918.537} C_VEL
LIN {X 0,Y 326.64,Z 233.792,A -85,B 0,C 180,E1 -14922.463,E2 -14922.463} C_VEL
LIN {X 0,Y 326.755,Z 233.78,A -85,B 0,C 180,E1 -14926.308,E2 -14926.308} C_VEL
LIN {X 0,Y 326.774,Z 233.779,A -85,B 0,C 180,E1 -14930.086,E2 -14930.086} C_VEL
LIN {X 0,Y 326.933,Z 233.758,A -85,B 0,C 180,E1 -14933.823,E2 -14933.823} C_VEL
LIN {X 0,Y 327.033,Z 233.743,A -85,B 0,C 180,E1 -14938.762,E2 -14938.762} C_VEL
LIN {X 0,Y 327.001,Z 233.749,A -85,B 0,C 180,E1 -14942.456,E2 -14942.456} C_VEL
LIN {X 0,Y 326.903,Z 233.761,A -85,B 0,C 180,E1 -14946.473,E2 -14946.473} C_VEL
LIN {X 0,Y 326.765,Z 233.78,A -85,B 0,C 180,E1 -14949.9,E2 -14949.9} C_VEL
LIN {X 0,Y 326.737,Z 233.785,A -85,B 0,C 180,E1 -14953.678,E2 -14953.678} C_VEL
LIN {X 0,Y 326.642,Z 233.797,A -85,B 0,C 180,E1 -14957.523,E2 -14957.523} C_VEL
LIN {X 0,Y 326.63,Z 233.795,A -85,B 0,C 180,E1 -14960.128,E2 -14960.128} C_VEL
LIN {X 0,Y 326.617,Z 233.797,A -85,B 0,C 180,E1 -14964.122,E2 -14964.122} C_VEL
LIN {X 0,Y 326.611,Z 233.796,A -85,B 0,C 180,E1 -14968.245,E2 -14968.245} C_VEL
LIN {X 0,Y 326.543,Z 233.806,A -85,B 0,C 180,E1 -14971.09,E2 -14971.09} C_VEL
LIN {X 0,Y 326.572,Z 233.801,A -85,B 0,C 180,E1 -14974.013,E2 -14974.013} C_VEL
LIN {X 0,Y 326.59,Z 233.805,A -85,B 0,C 180,E1 -14977.232,E2 -14977.232} C_VEL
LIN {X 0,Y 326.538,Z 233.811,A -85,B 0,C 180,E1 -14981.125,E2 -14981.125} C_VEL
LIN {X 0,Y 326.512,Z 233.811,A -85,B 0,C 180,E1 -14984.742,E2 -14984.742} C_VEL
LIN {X 0,Y 326.531,Z 233.808,A -85,B 0,C 180,E1 -14988.148,E2 -14988.148} C_VEL
LIN {X 0,Y 326.576,Z 233.806,A -85,B 0,C 180,E1 -14991.386,E2 -14991.386} C_VEL
LIN {X 0,Y 326.57,Z 233.805,A -85,B 0,C 180,E1 -14994.847,E2 -14994.847} C_VEL
LIN {X 0,Y 326.557,Z 233.808,A -85,B 0,C 180,E1 -14997.451,E2 -14997.451} C_VEL
LIN {X 0,Y 326.609,Z 233.798,A -85,B 0,C 180,E1 -15000.337,E2 -15000.337} C_VEL
LIN {X 0,Y 326.64,Z 233.795,A -85,B 0,C 180,E1 -15004.513,E2 -15004.513} C_VEL
LIN {X 0,Y 326.617,Z 233.798,A -85,B 0,C 180,E1 -15008.544,E2 -15008.544} C_VEL
LIN {X 0,Y 326.689,Z 233.794,A -85,B 0,C 180,E1 -15011.175,E2 -15011.175} C_VEL
LIN {X 0,Y 326.706,Z 233.788,A -85,B 0,C 180,E1 -15015.431,E2 -15015.431} C_VEL
LIN {X 0,Y 326.715,Z 233.788,A -85,B 0,C 180,E1 -15018.837,E2 -15018.837} C_VEL
LIN {X 0,Y 326.927,Z 233.76,A -85,B 0,C 180,E1 -15022.589,E2 -15022.589} C_VEL
LIN {X 0,Y 326.729,Z 233.789,A -85,B 0,C 180,E1 -15025.064,E2 -15025.064} C_VEL
LIN {X 0,Y 327.017,Z 233.749,A -85,B 0,C 180,E1 -15027.537,E2 -15027.537} C_VEL
LIN {X 0,Y 327.158,Z 233.729,A -85,B 0,C 180,E1 -15030,E2 -15030} C_VEL
LIN {X 0,Y 327.017,Z 233.748,A -85,B 0,C 180,E1 -15032.463,E2 -15032.463} C_VEL
LIN {X 0,Y 326.931,Z 233.844,A -85,B 0,C 180,E1 -15037.216,E2 -15037.216} C_VEL
LIN {X 0,Y 328.013,Z 240.07,A -85,B 0,C 180,E1 -15039.115,E2 -15039.115} C_VEL
LIN {X 0,Y 334.4,Z 258.549,A -85,B 0,C 180,E1 -15039.991,E2 -15039.991} C_VEL
LIN {X 0,Y 336.392,Z 268.888,A -85,B 0,C 180,E1 -15040.366,E2 -15040.366} C_VEL
LIN {X 0,Y 334.509,Z 347.124,A -85,B 0,C 180,E1 -15042.128,E2 -15042.128} C_VEL
LIN {X 0,Y 333.857,Z 360.324,A -85,B 0,C 180,E1 -15042.653,E2 -15042.653} C_VEL
LIN {X 0,Y 333.119,Z 373.148,A -85,B 0,C 180,E1 -15043.419,E2 -15043.419} C_VEL
LIN {X 0,Y 332.246,Z 384.26,A -85,B 0,C 180,E1 -15044.309,E2 -15044.309} C_VEL
LIN {X 0,Y 331.086,Z 396.169,A -85,B 0,C 180,E1 -15045.544,E2 -15045.544} C_VEL
LIN {X 0,Y 329.898,Z 406.752,A -85,B 0,C 180,E1 -15046.926,E2 -15046.926} C_VEL
LIN {X 0,Y 328.724,Z 415.78,A -85,B 0,C 180,E1 -15048.381,E2 -15048.381} C_VEL
LIN {X 0,Y 327.725,Z 424.214,A -85,B 0,C 180,E1 -15050.066,E2 -15050.066} C_VEL
LIN {X 0,Y 326.834,Z 431.571,A -85,B 0,C 180,E1 -15051.881,E2 -15051.881} C_VEL
LIN {X 0,Y 326.222,Z 436.865,A -85,B 0,C 180,E1 -15053.487,E2 -15053.487} C_VEL
LIN {X 0,Y 325.608,Z 442.315,A -85,B 0,C 180,E1 -15055.574,E2 -15055.574} C_VEL
LIN {X 0,Y 325.295,Z 446.373,A -85,B 0,C 180,E1 -15057.671,E2 -15057.671} C_VEL
LIN {X 0,Y 324.821,Z 449.425,A -85,B 0,C 180,E1 -15060.084,E2 -15060.084} C_VEL
LIN {X 0,Y 324.658,Z 450.919,A -85,B 0,C 180,E1 -15062.427,E2 -15062.427} C_VEL
LIN {X 0,Y 324.722,Z 450.997,A -85,B 0,C 180,E1 -15064.688,E2 -15064.688} C_VEL
LIN {X 0,Y 324.95,Z 449.795,A -85,B 0,C 180,E1 -15066.864,E2 -15066.864} C_VEL
LIN {X 0,Y 325.328,Z 447.452,A -85,B 0,C 180,E1 -15068.965,E2 -15068.965} C_VEL
LIN {X 0,Y 325.918,Z 443.974,A -85,B 0,C 180,E1 -15071.013,E2 -15071.013} C_VEL
LIN {X 0,Y 326.622,Z 439.382,A -85,B 0,C 180,E1 -15072.995,E2 -15072.995} C_VEL
LIN {X 0,Y 327.591,Z 433.101,A -85,B 0,C 180,E1 -15075.068,E2 -15075.068} C_VEL
LIN {X 0,Y 328.729,Z 426.234,A -85,B 0,C 180,E1 -15076.845,E2 -15076.845} C_VEL
LIN {X 0,Y 329.557,Z 421.297,A -85,B 0,C 180,E1 -15077.918,E2 -15077.918} C_VEL
LIN {X 0,Y 329.571,Z 417.492,A -85,B 0,C 180,E1 -15078.701,E2 -15078.701} C_VEL
LIN {X 0,Y 327.849,Z 411.087,A -85,B 0,C 180,E1 -15079.988,E2 -15079.988} C_VEL
LIN {X 0,Y 326.156,Z 404.266,A -85,B 0,C 180,E1 -15081.211,E2 -15081.211} C_VEL
LIN {X 0,Y 326.178,Z 399.666,A -85,B 0,C 180,E1 -15081.868,E2 -15081.868} C_VEL
LIN {X 0,Y 327.6,Z 388.762,A -85,B 0,C 180,E1 -15083.092,E2 -15083.092} C_VEL
LIN {X 0,Y 328.925,Z 376.351,A -85,B 0,C 180,E1 -15084.178,E2 -15084.178} C_VEL
LIN {X 0,Y 330.004,Z 363.569,A -85,B 0,C 180,E1 -15085.002,E2 -15085.002} C_VEL
LIN {X 0,Y 330.762,Z 350.767,A -85,B 0,C 180,E1 -15085.563,E2 -15085.563} C_VEL
LIN {X 0,Y 331.446,Z 330.086,A -85,B 0,C 180,E1 -15086.089,E2 -15086.089} C_VEL
LIN {X 0,Y 333.082,Z 270.529,A -85,B 0,C 180,E1 -15087.471,E2 -15087.471} C_VEL
LIN {X 0,Y 331.723,Z 264.938,A -85,B 0,C 180,E1 -15087.742,E2 -15087.742} C_VEL
LIN {X 0,Y 325.259,Z 249.901,A -85,B 0,C 180,E1 -15088.773,E2 -15088.773} C_VEL
LIN {X 0,Y 321.141,Z 240.964,A -85,B 0,C 180,E1 -15089.471,E2 -15089.471} C_VEL
LIN {X 0,Y 319.599,Z 234.677,A -85,B 0,C 180,E1 -15091.592,E2 -15091.592} C_VEL
LIN {X 0,Y 319.577,Z 234.678,A -85,B 0,C 180,E1 -15095.311,E2 -15095.311} C_VEL
LIN {X 0,Y 319.571,Z 234.677,A -85,B 0,C 180,E1 -15098.055,E2 -15098.055} C_VEL
LIN {X 0,Y 319.666,Z 234.669,A -85,B 0,C 180,E1 -15100.97,E2 -15100.97} C_VEL
LIN {X 0,Y 319.711,Z 234.658,A -85,B 0,C 180,E1 -15105.283,E2 -15105.283} C_VEL
LIN {X 0,Y 319.736,Z 234.657,A -85,B 0,C 180,E1 -15109.88,E2 -15109.88} C_VEL
LIN {X 0,Y 319.902,Z 234.635,A -85,B 0,C 180,E1 -15113.701,E2 -15113.701} C_VEL
LIN {X 0,Y 319.976,Z 234.623,A -85,B 0,C 180,E1 -15117.49,E2 -15117.49} C_VEL
LIN {X 0,Y 320.102,Z 234.61,A -85,B 0,C 180,E1 -15120.007,E2 -15120.007} C_VEL
LIN {X 0,Y 319.95,Z 234.623,A -85,B 0,C 180,E1 -15122.525,E2 -15122.525} C_VEL
LIN {X 0,Y 319.909,Z 234.626,A -85,B 0,C 180,E1 -15126.313,E2 -15126.313} C_VEL
LIN {X 0,Y 319.732,Z 234.648,A -85,B 0,C 180,E1 -15130.135,E2 -15130.135} C_VEL
LIN {X 0,Y 319.73,Z 234.65,A -85,B 0,C 180,E1 -15133.999,E2 -15133.999} C_VEL
LIN {X 0,Y 319.615,Z 234.667,A -85,B 0,C 180,E1 -15137.936,E2 -15137.936} C_VEL
LIN {X 0,Y 319.567,Z 234.673,A -85,B 0,C 180,E1 -15141.961,E2 -15141.961} C_VEL
LIN {X 0,Y 319.554,Z 234.673,A -85,B 0,C 180,E1 -15146.101,E2 -15146.101} C_VEL
LIN {X 0,Y 319.53,Z 234.68,A -85,B 0,C 180,E1 -15148.946,E2 -15148.946} C_VEL
LIN {X 0,Y 319.526,Z 234.683,A -85,B 0,C 180,E1 -15151.869,E2 -15151.869} C_VEL
LIN {X 0,Y 319.586,Z 234.675,A -85,B 0,C 180,E1 -15155.547,E2 -15155.547} C_VEL
LIN {X 0,Y 319.526,Z 234.68,A -85,B 0,C 180,E1 -15159.639,E2 -15159.639} C_VEL
LIN {X 0,Y 319.497,Z 234.691,A -85,B 0,C 180,E1 -15163.458,E2 -15163.458} C_VEL
LIN {X 0,Y 319.498,Z 234.689,A -85,B 0,C 180,E1 -15167.009,E2 -15167.009} C_VEL
LIN {X 0,Y 319.529,Z 234.686,A -85,B 0,C 180,E1 -15170.37,E2 -15170.37} C_VEL
LIN {X 0,Y 319.592,Z 234.678,A -85,B 0,C 180,E1 -15174.462,E2 -15174.462} C_VEL
LIN {X 0,Y 319.586,Z 234.753,A -85,B 0,C 180,E1 -15176.225,E2 -15176.225} C_VEL
LIN {X 0,Y 322.207,Z 245.329,A -85,B 0,C 180,E1 -15179.547,E2 -15179.547} C_VEL
LIN {X 0,Y 324.596,Z 256.999,A -85,B 0,C 180,E1 -15182.956,E2 -15182.956} C_VEL
LIN {X 0,Y 324.833,Z 260.768,A -85,B 0,C 180,E1 -15183.974,E2 -15183.974} C_VEL
LIN {X 0,Y 329.577,Z 284.451,A -85,B 0,C 180,E1 -15185.072,E2 -15185.072} C_VEL
LIN {X 0,Y 332.31,Z 303.236,A -85,B 0,C 180,E1 -15185.805,E2 -15185.805} C_VEL
LIN {X 0,Y 330.441,Z 370.532,A -85,B 0,C 180,E1 -15187.392,E2 -15187.392} C_VEL
LIN {X 0,Y 329.426,Z 384.321,A -85,B 0,C 180,E1 -15187.955,E2 -15187.955} C_VEL
LIN {X 0,Y 328.222,Z 397.047,A -85,B 0,C 180,E1 -15188.736,E2 -15188.736} C_VEL
LIN {X 0,Y 326.832,Z 408.744,A -85,B 0,C 180,E1 -15189.712,E2 -15189.712} C_VEL
LIN {X 0,Y 325.201,Z 420.081,A -85,B 0,C 180,E1 -15190.922,E2 -15190.922} C_VEL
LIN {X 0,Y 323.664,Z 430.346,A -85,B 0,C 180,E1 -15192.303,E2 -15192.303} C_VEL
LIN {X 0,Y 322.149,Z 440.437,A -85,B 0,C 180,E1 -15194.017,E2 -15194.017} C_VEL
LIN {X 0,Y 320.879,Z 448.632,A -85,B 0,C 180,E1 -15195.736,E2 -15195.736} C_VEL
LIN {X 0,Y 319.577,Z 455.938,A -85,B 0,C 180,E1 -15197.619,E2 -15197.619} C_VEL
LIN {X 0,Y 318.906,Z 460.886,A -85,B 0,C 180,E1 -15199.204,E2 -15199.204} C_VEL
LIN {X 0,Y 318.344,Z 465.711,A -85,B 0,C 180,E1 -15201.11,E2 -15201.11} C_VEL
LIN {X 0,Y 317.943,Z 469.416,A -85,B 0,C 180,E1 -15203.017,E2 -15203.017} C_VEL
LIN {X 0,Y 317.794,Z 472.106,A -85,B 0,C 180,E1 -15204.925,E2 -15204.925} C_VEL
LIN {X 0,Y 317.808,Z 473.387,A -85,B 0,C 180,E1 -15206.196,E2 -15206.196} C_VEL
LIN {X 0,Y 317.786,Z 474.236,A -85,B 0,C 180,E1 -15207.465,E2 -15207.465} C_VEL
LIN {X 0,Y 317.78,Z 474.661,A -85,B 0,C 180,E1 -15208.733,E2 -15208.733} C_VEL
LIN {X 0,Y 317.833,Z 474.695,A -85,B 0,C 180,E1 -15210,E2 -15210} C_VEL
LIN {X 0,Y 317.792,Z 474.333,A -85,B 0,C 180,E1 -15211.267,E2 -15211.267} C_VEL
LIN {X 0,Y 317.791,Z 473.545,A -85,B 0,C 180,E1 -15212.535,E2 -15212.535} C_VEL
LIN {X 0,Y 317.821,Z 472.319,A -85,B 0,C 180,E1 -15213.804,E2 -15213.804} C_VEL
LIN {X 0,Y 317.86,Z 469.684,A -85,B 0,C 180,E1 -15215.713,E2 -15215.713} C_VEL
LIN {X 0,Y 318.054,Z 466.017,A -85,B 0,C 180,E1 -15217.619,E2 -15217.619} C_VEL
LIN {X 0,Y 318.439,Z 461.203,A -85,B 0,C 180,E1 -15219.528,E2 -15219.528} C_VEL
LIN {X 0,Y 318.993,Z 455.097,A -85,B 0,C 180,E1 -15221.437,E2 -15221.437} C_VEL
LIN {X 0,Y 320.01,Z 447.501,A -85,B 0,C 180,E1 -15223.332,E2 -15223.332} C_VEL
LIN {X 0,Y 320.995,Z 439.73,A -85,B 0,C 180,E1 -15224.907,E2 -15224.907} C_VEL
LIN {X 0,Y 322.095,Z 430.234,A -85,B 0,C 180,E1 -15226.478,E2 -15226.478} C_VEL
LIN {X 0,Y 323.325,Z 419.69,A -85,B 0,C 180,E1 -15227.88,E2 -15227.88} C_VEL
LIN {X 0,Y 324.608,Z 407.984,A -85,B 0,C 180,E1 -15229.115,E2 -15229.115} C_VEL
LIN {X 0,Y 325.835,Z 395.542,A -85,B 0,C 180,E1 -15230.106,E2 -15230.106} C_VEL
LIN {X 0,Y 326.862,Z 382.517,A -85,B 0,C 180,E1 -15230.861,E2 -15230.861} C_VEL
LIN {X 0,Y 327.533,Z 369.814,A -85,B 0,C 180,E1 -15231.352,E2 -15231.352} C_VEL
LIN {X 0,Y 329.029,Z 301.738,A -85,B 0,C 180,E1 -15232.926,E2 -15232.926} C_VEL
LIN {X 0,Y 323.209,Z 262.429,A -85,B 0,C 180,E1 -15234.29,E2 -15234.29} C_VEL
LIN {X 0,Y 323.775,Z 255.549,A -85,B 0,C 180,E1 -15236.056,E2 -15236.056} C_VEL
LIN {X 0,Y 321.719,Z 244.727,A -85,B 0,C 180,E1 -15239.088,E2 -15239.088} C_VEL
LIN {X 0,Y 319.566,Z 234.68,A -85,B 0,C 180,E1 -15242.043,E2 -15242.043} C_VEL
LIN {X 0,Y 319.584,Z 234.677,A -85,B 0,C 180,E1 -15245.537,E2 -15245.537} C_VEL
LIN {X 0,Y 319.53,Z 234.684,A -85,B 0,C 180,E1 -15249.63,E2 -15249.63} C_VEL
LIN {X 0,Y 319.483,Z 234.689,A -85,B 0,C 180,E1 -15253.447,E2 -15253.447} C_VEL
LIN {X 0,Y 319.495,Z 234.685,A -85,B 0,C 180,E1 -15257,E2 -15257} C_VEL
LIN {X 0,Y 319.527,Z 234.681,A -85,B 0,C 180,E1 -15260.361,E2 -15260.361} C_VEL
LIN {X 0,Y 319.586,Z 234.673,A -85,B 0,C 180,E1 -15264.454,E2 -15264.454} C_VEL
LIN {X 0,Y 319.525,Z 234.682,A -85,B 0,C 180,E1 -15268.131,E2 -15268.131} C_VEL
LIN {X 0,Y 319.549,Z 234.683,A -85,B 0,C 180,E1 -15271.608,E2 -15271.608} C_VEL
LIN {X 0,Y 319.546,Z 234.68,A -85,B 0,C 180,E1 -15275.293,E2 -15275.293} C_VEL
LIN {X 0,Y 319.567,Z 234.676,A -85,B 0,C 180,E1 -15278.039,E2 -15278.039} C_VEL
LIN {X 0,Y 319.593,Z 234.67,A -85,B 0,C 180,E1 -15282.063,E2 -15282.063} C_VEL
LIN {X 0,Y 319.73,Z 234.656,A -85,B 0,C 180,E1 -15286.001,E2 -15286.001} C_VEL
LIN {X 0,Y 319.727,Z 234.658,A -85,B 0,C 180,E1 -15289.865,E2 -15289.865} C_VEL
LIN {X 0,Y 319.891,Z 234.636,A -85,B 0,C 180,E1 -15293.687,E2 -15293.687} C_VEL
LIN {X 0,Y 320,Z 234.618,A -85,B 0,C 180,E1 -15298.734,E2 -15298.734} C_VEL
LIN {X 0,Y 319.947,Z 234.627,A -85,B 0,C 180,E1 -15302.511,E2 -15302.511} C_VEL
LIN {X 0,Y 319.867,Z 234.637,A -85,B 0,C 180,E1 -15306.455,E2 -15306.455} C_VEL
LIN {X 0,Y 319.718,Z 234.656,A -85,B 0,C 180,E1 -15310.121,E2 -15310.121} C_VEL
LIN {X 0,Y 319.712,Z 234.658,A -85,B 0,C 180,E1 -15313.985,E2 -15313.985} C_VEL
LIN {X 0,Y 319.603,Z 234.67,A -85,B 0,C 180,E1 -15317.922,E2 -15317.922} C_VEL
LIN {X 0,Y 319.582,Z 234.673,A -85,B 0,C 180,E1 -15320.592,E2 -15320.592} C_VEL
LIN {X 0,Y 319.541,Z 234.683,A -85,B 0,C 180,E1 -15323.312,E2 -15323.312} C_VEL
LIN {X 0,Y 319.56,Z 234.675,A -85,B 0,C 180,E1 -15326.085,E2 -15326.085} C_VEL
LIN {X 0,Y 319.537,Z 234.678,A -85,B 0,C 180,E1 -15328.929,E2 -15328.929} C_VEL
LIN {X 0,Y 319.492,Z 234.681,A -85,B 0,C 180,E1 -15331.856,E2 -15331.856} C_VEL
LIN {X 0,Y 319.544,Z 234.681,A -85,B 0,C 180,E1 -15335.536,E2 -15335.536} C_VEL
LIN {X 0,Y 319.521,Z 234.683,A -85,B 0,C 180,E1 -15339.662,E2 -15339.662} C_VEL
LIN {X 0,Y 319.515,Z 234.685,A -85,B 0,C 180,E1 -15343.461,E2 -15343.461} C_VEL
LIN {X 0,Y 319.517,Z 234.685,A -85,B 0,C 180,E1 -15347.012,E2 -15347.012} C_VEL
LIN {X 0,Y 319.5,Z 234.683,A -85,B 0,C 180,E1 -15350.365,E2 -15350.365} C_VEL
LIN {X 0,Y 319.51,Z 234.685,A -85,B 0,C 180,E1 -15353.567,E2 -15353.567} C_VEL
LIN {X 0,Y 319.528,Z 234.681,A -85,B 0,C 180,E1 -15356.682,E2 -15356.682} C_VEL
LIN {X 0,Y 319.54,Z 234.681,A -85,B 0,C 180,E1 -15359.612,E2 -15359.612} C_VEL
LIN {X 0,Y 319.556,Z 234.677,A -85,B 0,C 180,E1 -15362.494,E2 -15362.494} C_VEL
LIN {X 0,Y 319.572,Z 234.68,A -85,B 0,C 180,E1 -15365.302,E2 -15365.302} C_VEL
LIN {X 0,Y 319.568,Z 234.675,A -85,B 0,C 180,E1 -15368.046,E2 -15368.046} C_VEL
LIN {X 0,Y 319.637,Z 234.671,A -85,B 0,C 180,E1 -15370.958,E2 -15370.958} C_VEL
LIN {X 0,Y 319.674,Z 234.666,A -85,B 0,C 180,E1 -15375.274,E2 -15375.274} C_VEL
LIN {X 0,Y 319.701,Z 234.659,A -85,B 0,C 180,E1 -15379.871,E2 -15379.871} C_VEL
LIN {X 0,Y 319.879,Z 234.637,A -85,B 0,C 180,E1 -15382.425,E2 -15382.425} C_VEL
LIN {X 0,Y 319.698,Z 234.664,A -85,B 0,C 180,E1 -15384.955,E2 -15384.955} C_VEL
LIN {X 0,Y 319.958,Z 234.629,A -85,B 0,C 180,E1 -15387.482,E2 -15387.482} C_VEL
LIN {X 0,Y 320.11,Z 234.608,A -85,B 0,C 180,E1 -15390,E2 -15390} C_VEL
LIN {X 0,Y 319.958,Z 234.628,A -85,B 0,C 180,E1 -15392.518,E2 -15392.518} C_VEL
LIN {X 0,Y 319.872,Z 234.68,A -85,B 0,C 180,E1 -15396.861,E2 -15396.861} C_VEL
LIN {X 0,Y 320.981,Z 240.573,A -85,B 0,C 180,E1 -15398.638,E2 -15398.638} C_VEL
LIN {X 0,Y 327.909,Z 260.34,A -85,B 0,C 180,E1 -15399.61,E2 -15399.61} C_VEL
LIN {X 0,Y 329.716,Z 270.586,A -85,B 0,C 180,E1 -15399.981,E2 -15399.981} C_VEL
LIN {X 0,Y 327.774,Z 347.58,A -85,B 0,C 180,E1 -15401.753,E2 -15401.753} C_VEL
LIN {X 0,Y 327.095,Z 360.721,A -85,B 0,C 180,E1 -15402.289,E2 -15402.289} C_VEL
LIN {X 0,Y 326.32,Z 373.517,A -85,B 0,C 180,E1 -15403.069,E2 -15403.069} C_VEL
LIN {X 0,Y 325.321,Z 385.507,A -85,B 0,C 180,E1 -15404.065,E2 -15404.065} C_VEL
LIN {X 0,Y 324.221,Z 396.487,A -85,B 0,C 180,E1 -15405.237,E2 -15405.237} C_VEL
LIN {X 0,Y 322.989,Z 407.029,A -85,B 0,C 180,E1 -15406.643,E2 -15406.643} C_VEL
LIN {X 0,Y 321.772,Z 416.084,A -85,B 0,C 180,E1 -15408.134,E2 -15408.134} C_VEL
LIN {X 0,Y 320.66,Z 425.349,A -85,B 0,C 180,E1 -15410.048,E2 -15410.048} C_VEL
LIN {X 0,Y 319.726,Z 432.7,A -85,B 0,C 180,E1 -15411.942,E2 -15411.942} C_VEL
LIN {X 0,Y 318.934,Z 439.139,A -85,B 0,C 180,E1 -15414.057,E2 -15414.057} C_VEL
LIN {X 0,Y 318.405,Z 444.085,A -85,B 0,C 180,E1 -15416.196,E2 -15416.196} C_VEL
LIN {X 0,Y 318.148,Z 447.114,A -85,B 0,C 180,E1 -15417.94,E2 -15417.94} C_VEL
LIN {X 0,Y 317.689,Z 449.972,A -85,B 0,C 180,E1 -15420.391,E2 -15420.391} C_VEL
LIN {X 0,Y 317.582,Z 451.272,A -85,B 0,C 180,E1 -15422.78,E2 -15422.78} C_VEL
LIN {X 0,Y 317.661,Z 451.145,A -85,B 0,C 180,E1 -15425.114,E2 -15425.114} C_VEL
LIN {X 0,Y 317.929,Z 449.823,A -85,B 0,C 180,E1 -15427.285,E2 -15427.285} C_VEL
LIN {X 0,Y 318.48,Z 446.82,A -85,B 0,C 180,E1 -15429.787,E2 -15429.787} C_VEL
LIN {X 0,Y 319.201,Z 442.255,A -85,B 0,C 180,E1 -15432.195,E2 -15432.195} C_VEL
LIN {X 0,Y 320.041,Z 437.638,A -85,B 0,C 180,E1 -15434.005,E2 -15434.005} C_VEL
LIN {X 0,Y 320.984,Z 431.903,A -85,B 0,C 180,E1 -15435.804,E2 -15435.804} C_VEL
LIN {X 0,Y 322.385,Z 423.786,A -85,B 0,C 180,E1 -15437.832,E2 -15437.832} C_VEL
LIN {X 0,Y 323.921,Z 414.528,A -85,B 0,C 180,E1 -15439.647,E2 -15439.647} C_VEL
LIN {X 0,Y 325.564,Z 404.272,A -85,B 0,C 180,E1 -15441.254,E2 -15441.254} C_VEL
LIN {X 0,Y 326.178,Z 399.666,A -85,B 0,C 180,E1 -15441.868,E2 -15441.868} C_VEL
LIN {X 0,Y 326.223,Z 394.956,A -85,B 0,C 180,E1 -15442.498,E2 -15442.498} C_VEL
LIN {X 0,Y 324.575,Z 387.144,A -85,B 0,C 180,E1 -15443.539,E2 -15443.539} C_VEL
LIN {X 0,Y 322.862,Z 378.929,A -85,B 0,C 180,E1 -15444.468,E2 -15444.468} C_VEL
LIN {X 0,Y 322.782,Z 373.594,A -85,B 0,C 180,E1 -15444.913,E2 -15444.913} C_VEL
LIN {X 0,Y 323.854,Z 359.969,A -85,B 0,C 180,E1 -15445.732,E2 -15445.732} C_VEL
LIN {X 0,Y 324.578,Z 347.012,A -85,B 0,C 180,E1 -15446.234,E2 -15446.234} C_VEL
LIN {X 0,Y 326.834,Z 271.83,A -85,B 0,C 180,E1 -15448.029,E2 -15448.029} C_VEL
LIN {X 0,Y 325.623,Z 267.26,A -85,B 0,C 180,E1 -15448.269,E2 -15448.269} C_VEL
LIN {X 0,Y 319.701,Z 253.422,A -85,B 0,C 180,E1 -15449.246,E2 -15449.246} C_VEL
LIN {X 0,Y 314.016,Z 241.317,A -85,B 0,C 180,E1 -15450.237,E2 -15450.237} C_VEL
LIN {X 0,Y 312.554,Z 235.551,A -85,B 0,C 180,E1 -15452.198,E2 -15452.198} C_VEL
LIN {X 0,Y 312.557,Z 235.553,A -85,B 0,C 180,E1 -15454.718,E2 -15454.718} C_VEL
LIN {X 0,Y 312.562,Z 235.551,A -85,B 0,C 180,E1 -15457.536,E2 -15457.536} C_VEL
LIN {X 0,Y 312.616,Z 235.547,A -85,B 0,C 180,E1 -15461.664,E2 -15461.664} C_VEL
LIN {X 0,Y 312.675,Z 235.534,A -85,B 0,C 180,E1 -15465.694,E2 -15465.694} C_VEL
LIN {X 0,Y 312.682,Z 235.536,A -85,B 0,C 180,E1 -15469.649,E2 -15469.649} C_VEL
LIN {X 0,Y 312.861,Z 235.512,A -85,B 0,C 180,E1 -15473.559,E2 -15473.559} C_VEL
LIN {X 0,Y 312.922,Z 235.502,A -85,B 0,C 180,E1 -15477.433,E2 -15477.433} C_VEL
LIN {X 0,Y 313.057,Z 235.488,A -85,B 0,C 180,E1 -15480.007,E2 -15480.007} C_VEL
LIN {X 0,Y 312.899,Z 235.501,A -85,B 0,C 180,E1 -15482.582,E2 -15482.582} C_VEL
LIN {X 0,Y 312.853,Z 235.506,A -85,B 0,C 180,E1 -15486.456,E2 -15486.456} C_VEL
LIN {X 0,Y 312.747,Z 235.522,A -85,B 0,C 180,E1 -15489.057,E2 -15489.057} C_VEL
LIN {X 0,Y 312.631,Z 235.539,A -85,B 0,C 180,E1 -15492.998,E2 -15492.998} C_VEL
LIN {X 0,Y 312.622,Z 235.541,A -85,B 0,C 180,E1 -15495.657,E2 -15495.657} C_VEL
LIN {X 0,Y 312.539,Z 235.55,A -85,B 0,C 180,E1 -15499.719,E2 -15499.719} C_VEL
LIN {X 0,Y 312.52,Z 235.548,A -85,B 0,C 180,E1 -15502.782,E2 -15502.782} C_VEL
LIN {X 0,Y 312.487,Z 235.553,A -85,B 0,C 180,E1 -15506.738,E2 -15506.738} C_VEL
LIN {X 0,Y 312.474,Z 235.556,A -85,B 0,C 180,E1 -15509.664,E2 -15509.664} C_VEL
LIN {X 0,Y 312.528,Z 235.548,A -85,B 0,C 180,E1 -15513.694,E2 -15513.694} C_VEL
LIN {X 0,Y 312.518,Z 235.554,A -85,B 0,C 180,E1 -15517.393,E2 -15517.393} C_VEL
LIN {X 0,Y 312.438,Z 235.569,A -85,B 0,C 180,E1 -15520.724,E2 -15520.724} C_VEL
LIN {X 0,Y 312.45,Z 235.57,A -85,B 0,C 180,E1 -15524.217,E2 -15524.217} C_VEL
LIN {X 0,Y 312.439,Z 235.571,A -85,B 0,C 180,E1 -15527.935,E2 -15527.935} C_VEL
LIN {X 0,Y 312.489,Z 235.563,A -85,B 0,C 180,E1 -15531.929,E2 -15531.929} C_VEL
LIN {X 0,Y 312.552,Z 235.598,A -85,B 0,C 180,E1 -15535.553,E2 -15535.553} C_VEL
LIN {X 0,Y 315.336,Z 246.702,A -85,B 0,C 180,E1 -15539.163,E2 -15539.163} C_VEL
LIN {X 0,Y 317.635,Z 258.093,A -85,B 0,C 180,E1 -15542.588,E2 -15542.588} C_VEL
LIN {X 0,Y 318.05,Z 260.596,A -85,B 0,C 180,E1 -15543.282,E2 -15543.282} C_VEL
LIN {X 0,Y 320.451,Z 270.471,A -85,B 0,C 180,E1 -15543.803,E2 -15543.803} C_VEL
LIN {X 0,Y 324.214,Z 291.158,A -85,B 0,C 180,E1 -15544.738,E2 -15544.738} C_VEL
LIN {X 0,Y 326.009,Z 304.922,A -85,B 0,C 180,E1 -15545.277,E2 -15545.277} C_VEL
LIN {X 0,Y 324.06,Z 370.211,A -85,B 0,C 180,E1 -15546.848,E2 -15546.848} C_VEL
LIN {X 0,Y 323.023,Z 383.819,A -85,B 0,C 180,E1 -15547.41,E2 -15547.41} C_VEL
LIN {X 0,Y 321.75,Z 396.619,A -85,B 0,C 180,E1 -15548.203,E2 -15548.203} C_VEL
LIN {X 0,Y 320.4,Z 407.561,A -85,B 0,C 180,E1 -15549.119,E2 -15549.119} C_VEL
LIN {X 0,Y 318.716,Z 419.062,A -85,B 0,C 180,E1 -15550.35,E2 -15550.35} C_VEL
LIN {X 0,Y 317.084,Z 429.465,A -85,B 0,C 180,E1 -15551.756,E2 -15551.756} C_VEL
LIN {X 0,Y 315.733,Z 437.998,A -85,B 0,C 180,E1 -15553.18,E2 -15553.18} C_VEL
LIN {X 0,Y 314.427,Z 445.894,A -85,B 0,C 180,E1 -15554.774,E2 -15554.774} C_VEL
LIN {X 0,Y 313.09,Z 453.628,A -85,B 0,C 180,E1 -15556.698,E2 -15556.698} C_VEL
LIN {X 0,Y 312.141,Z 458.946,A -85,B 0,C 180,E1 -15558.309,E2 -15558.309} C_VEL
LIN {X 0,Y 311.454,Z 464.115,A -85,B 0,C 180,E1 -15560.257,E2 -15560.257} C_VEL
LIN {X 0,Y 311.002,Z 468.151,A -85,B 0,C 180,E1 -15562.208,E2 -15562.208} C_VEL
LIN {X 0,Y 310.744,Z 471.415,A -85,B 0,C 180,E1 -15564.385,E2 -15564.385} C_VEL
LIN {X 0,Y 310.718,Z 473.174,A -85,B 0,C 180,E1 -15566.109,E2 -15566.109} C_VEL
LIN {X 0,Y 310.708,Z 473.994,A -85,B 0,C 180,E1 -15567.407,E2 -15567.407} C_VEL
LIN {X 0,Y 310.693,Z 474.404,A -85,B 0,C 180,E1 -15568.704,E2 -15568.704} C_VEL
LIN {X 0,Y 310.742,Z 474.424,A -85,B 0,C 180,E1 -15570,E2 -15570} C_VEL
LIN {X 0,Y 310.705,Z 474.046,A -85,B 0,C 180,E1 -15571.296,E2 -15571.296} C_VEL
LIN {X 0,Y 310.713,Z 473.227,A -85,B 0,C 180,E1 -15572.593,E2 -15572.593} C_VEL
LIN {X 0,Y 310.732,Z 471.984,A -85,B 0,C 180,E1 -15573.891,E2 -15573.891} C_VEL
LIN {X 0,Y 310.786,Z 469.564,A -85,B 0,C 180,E1 -15575.693,E2 -15575.693} C_VEL
LIN {X 0,Y 311.002,Z 465.61,A -85,B 0,C 180,E1 -15577.792,E2 -15577.792} C_VEL
LIN {X 0,Y 311.391,Z 460.753,A -85,B 0,C 180,E1 -15579.745,E2 -15579.745} C_VEL
LIN {X 0,Y 311.994,Z 454.602,A -85,B 0,C 180,E1 -15581.697,E2 -15581.697} C_VEL
LIN {X 0,Y 313.072,Z 446.955,A -85,B 0,C 180,E1 -15583.633,E2 -15583.633} C_VEL
LIN {X 0,Y 314.099,Z 439.116,A -85,B 0,C 180,E1 -15585.242,E2 -15585.242} C_VEL
LIN {X 0,Y 315.206,Z 429.514,A -85,B 0,C 180,E1 -15586.849,E2 -15586.849} C_VEL
LIN {X 0,Y 316.548,Z 418.881,A -85,B 0,C 180,E1 -15588.276,E2 -15588.276} C_VEL
LIN {X 0,Y 317.889,Z 407.011,A -85,B 0,C 180,E1 -15589.535,E2 -15589.535} C_VEL
LIN {X 0,Y 319.165,Z 394.331,A -85,B 0,C 180,E1 -15590.545,E2 -15590.545} C_VEL
LIN {X 0,Y 320.127,Z 381.73,A -85,B 0,C 180,E1 -15591.279,E2 -15591.279} C_VEL
LIN {X 0,Y 320.816,Z 368.547,A -85,B 0,C 180,E1 -15591.779,E2 -15591.779} C_VEL
LIN {X 0,Y 322.391,Z 302.932,A -85,B 0,C 180,E1 -15593.322,E2 -15593.322} C_VEL
LIN {X 0,Y 316.364,Z 262.189,A -85,B 0,C 180,E1 -15594.773,E2 -15594.773} C_VEL
LIN {X 0,Y 316.858,Z 257.56,A -85,B 0,C 180,E1 -15595.98,E2 -15595.98} C_VEL
LIN {X 0,Y 315.2,Z 248.188,A -85,B 0,C 180,E1 -15598.644,E2 -15598.644} C_VEL
LIN {X 0,Y 312.846,Z 237.018,A -85,B 0,C 180,E1 -15601.964,E2 -15601.964} C_VEL
LIN {X 0,Y 312.532,Z 235.555,A -85,B 0,C 180,E1 -15602.413,E2 -15602.413} C_VEL
LIN {X 0,Y 312.541,Z 235.554,A -85,B 0,C 180,E1 -15605.943,E2 -15605.943} C_VEL
LIN {X 0,Y 312.448,Z 235.566,A -85,B 0,C 180,E1 -15610.106,E2 -15610.106} C_VEL
LIN {X 0,Y 312.443,Z 235.566,A -85,B 0,C 180,E1 -15614.21,E2 -15614.21} C_VEL
LIN {X 0,Y 312.436,Z 235.567,A -85,B 0,C 180,E1 -15617.927,E2 -15617.927} C_VEL
LIN {X 0,Y 312.484,Z 235.562,A -85,B 0,C 180,E1 -15621.921,E2 -15621.921} C_VEL
LIN {X 0,Y 312.537,Z 235.553,A -85,B 0,C 180,E1 -15624.215,E2 -15624.215} C_VEL
LIN {X 0,Y 312.507,Z 235.558,A -85,B 0,C 180,E1 -15627.328,E2 -15627.328} C_VEL
LIN {X 0,Y 312.488,Z 235.56,A -85,B 0,C 180,E1 -15631.295,E2 -15631.295} C_VEL
LIN {X 0,Y 312.527,Z 235.552,A -85,B 0,C 180,E1 -15634.699,E2 -15634.699} C_VEL
LIN {X 0,Y 312.544,Z 235.555,A -85,B 0,C 180,E1 -15637.519,E2 -15637.519} C_VEL
LIN {X 0,Y 312.551,Z 235.548,A -85,B 0,C 180,E1 -15641.645,E2 -15641.645} C_VEL
LIN {X 0,Y 312.684,Z 235.537,A -85,B 0,C 180,E1 -15645.679,E2 -15645.679} C_VEL
LIN {X 0,Y 312.678,Z 235.538,A -85,B 0,C 180,E1 -15649.634,E2 -15649.634} C_VEL
LIN {X 0,Y 312.833,Z 235.515,A -85,B 0,C 180,E1 -15653.544,E2 -15653.544} C_VEL
LIN {X 0,Y 312.967,Z 235.492,A -85,B 0,C 180,E1 -15658.706,E2 -15658.706} C_VEL
LIN {X 0,Y 312.895,Z 235.506,A -85,B 0,C 180,E1 -15662.567,E2 -15662.567} C_VEL
LIN {X 0,Y 312.823,Z 235.515,A -85,B 0,C 180,E1 -15666.442,E2 -15666.442} C_VEL
LIN {X 0,Y 312.736,Z 235.527,A -85,B 0,C 180,E1 -15669.043,E2 -15669.043} C_VEL
LIN {X 0,Y 312.613,Z 235.543,A -85,B 0,C 180,E1 -15672.984,E2 -15672.984} C_VEL
LIN {X 0,Y 312.602,Z 235.546,A -85,B 0,C 180,E1 -15675.643,E2 -15675.643} C_VEL
LIN {X 0,Y 312.554,Z 235.551,A -85,B 0,C 180,E1 -15679.703,E2 -15679.703} C_VEL
LIN {X 0,Y 312.517,Z 235.554,A -85,B 0,C 180,E1 -15682.78,E2 -15682.78} C_VEL
LIN {X 0,Y 312.492,Z 235.556,A -85,B 0,C 180,E1 -15686.721,E2 -15686.721} C_VEL
LIN {X 0,Y 312.493,Z 235.553,A -85,B 0,C 180,E1 -15689.645,E2 -15689.645} C_VEL
LIN {X 0,Y 312.486,Z 235.556,A -85,B 0,C 180,E1 -15693.682,E2 -15693.682} C_VEL
LIN {X 0,Y 312.483,Z 235.563,A -85,B 0,C 180,E1 -15697.379,E2 -15697.379} C_VEL
LIN {X 0,Y 312.451,Z 235.563,A -85,B 0,C 180,E1 -15700.703,E2 -15700.703} C_VEL
LIN {X 0,Y 312.43,Z 235.563,A -85,B 0,C 180,E1 -15704.2,E2 -15704.2} C_VEL
LIN {X 0,Y 312.441,Z 235.563,A -85,B 0,C 180,E1 -15707.913,E2 -15707.913} C_VEL
LIN {X 0,Y 312.458,Z 235.561,A -85,B 0,C 180,E1 -15711.912,E2 -15711.912} C_VEL
LIN {X 0,Y 312.483,Z 235.558,A -85,B 0,C 180,E1 -15714.215,E2 -15714.215} C_VEL
LIN {X 0,Y 312.455,Z 235.566,A -85,B 0,C 180,E1 -15717.329,E2 -15717.329} C_VEL
LIN {X 0,Y 312.501,Z 235.56,A -85,B 0,C 180,E1 -15721.272,E2 -15721.272} C_VEL
LIN {X 0,Y 312.541,Z 235.553,A -85,B 0,C 180,E1 -15724.708,E2 -15724.708} C_VEL
LIN {X 0,Y 312.562,Z 235.551,A -85,B 0,C 180,E1 -15727.528,E2 -15727.528} C_VEL
LIN {X 0,Y 312.584,Z 235.546,A -85,B 0,C 180,E1 -15731.653,E2 -15731.653} C_VEL
LIN {X 0,Y 312.637,Z 235.539,A -85,B 0,C 180,E1 -15735.684,E2 -15735.684} C_VEL
LIN {X 0,Y 312.646,Z 235.538,A -85,B 0,C 180,E1 -15739.64,E2 -15739.64} C_VEL
LIN {X 0,Y 312.817,Z 235.516,A -85,B 0,C 180,E1 -15742.253,E2 -15742.253} C_VEL
LIN {X 0,Y 312.668,Z 235.538,A -85,B 0,C 180,E1 -15744.842,E2 -15744.842} C_VEL
LIN {X 0,Y 312.902,Z 235.508,A -85,B 0,C 180,E1 -15747.425,E2 -15747.425} C_VEL
LIN {X 0,Y 313.062,Z 235.486,A -85,B 0,C 180,E1 -15750,E2 -15750} C_VEL
LIN {X 0,Y 312.902,Z 235.507,A -85,B 0,C 180,E1 -15752.575,E2 -15752.575} C_VEL
LIN {X 0,Y 312.877,Z 235.625,A -85,B 0,C 180,E1 -15756.529,E2 -15756.529} C_VEL
LIN {X 0,Y 313.841,Z 240.804,A -85,B 0,C 180,E1 -15758.126,E2 -15758.126} C_VEL
LIN {X 0,Y 321.529,Z 262.7,A -85,B 0,C 180,E1 -15759.234,E2 -15759.234} C_VEL
LIN {X 0,Y 323.075,Z 270.794,A -85,B 0,C 180,E1 -15759.543,E2 -15759.543} C_VEL
LIN {X 0,Y 321.053,Z 348.036,A -85,B 0,C 180,E1 -15761.362,E2 -15761.362} C_VEL
LIN {X 0,Y 320.309,Z 361.909,A -85,B 0,C 180,E1 -15761.95,E2 -15761.95} C_VEL
LIN {X 0,Y 319.483,Z 374.916,A -85,B 0,C 180,E1 -15762.784,E2 -15762.784} C_VEL
LIN {X 0,Y 318.415,Z 387.005,A -85,B 0,C 180,E1 -15763.838,E2 -15763.838} C_VEL
LIN {X 0,Y 317.214,Z 398.212,A -85,B 0,C 180,E1 -15765.089,E2 -15765.089} C_VEL
LIN {X 0,Y 316.012,Z 408.125,A -85,B 0,C 180,E1 -15766.472,E2 -15766.472} C_VEL
LIN {X 0,Y 314.624,Z 418.169,A -85,B 0,C 180,E1 -15768.223,E2 -15768.223} C_VEL
LIN {X 0,Y 313.579,Z 426.479,A -85,B 0,C 180,E1 -15770.027,E2 -15770.027} C_VEL
LIN {X 0,Y 312.694,Z 432.997,A -85,B 0,C 180,E1 -15771.767,E2 -15771.767} C_VEL
LIN {X 0,Y 311.876,Z 439.426,A -85,B 0,C 180,E1 -15773.929,E2 -15773.929} C_VEL
LIN {X 0,Y 311.333,Z 444.389,A -85,B 0,C 180,E1 -15776.127,E2 -15776.127} C_VEL
LIN {X 0,Y 310.948,Z 448.007,A -85,B 0,C 180,E1 -15778.335,E2 -15778.335} C_VEL
LIN {X 0,Y 310.555,Z 450.496,A -85,B 0,C 180,E1 -15780.708,E2 -15780.708} C_VEL
LIN {X 0,Y 310.477,Z 451.582,A -85,B 0,C 180,E1 -15783.138,E2 -15783.138} C_VEL
LIN {X 0,Y 310.603,Z 451.325,A -85,B 0,C 180,E1 -15785.473,E2 -15785.473} C_VEL
LIN {X 0,Y 310.906,Z 449.856,A -85,B 0,C 180,E1 -15787.721,E2 -15787.721} C_VEL
LIN {X 0,Y 311.445,Z 447.23,A -85,B 0,C 180,E1 -15789.909,E2 -15789.909} C_VEL
LIN {X 0,Y 312.065,Z 443.515,A -85,B 0,C 180,E1 -15792.011,E2 -15792.011} C_VEL
LIN {X 0,Y 313.016,Z 438.496,A -85,B 0,C 180,E1 -15794.108,E2 -15794.108} C_VEL
LIN {X 0,Y 314.086,Z 432.4,A -85,B 0,C 180,E1 -15796.093,E2 -15796.093} C_VEL
LIN {X 0,Y 315.477,Z 424.725,A -85,B 0,C 180,E1 -15798.075,E2 -15798.075} C_VEL
LIN {X 0,Y 316.972,Z 416.435,A -85,B 0,C 180,E1 -15799.784,E2 -15799.784} C_VEL
LIN {X 0,Y 318.49,Z 407.27,A -85,B 0,C 180,E1 -15801.314,E2 -15801.314} C_VEL
LIN {X 0,Y 320.072,Z 396.65,A -85,B 0,C 180,E1 -15802.744,E2 -15802.744} C_VEL
LIN {X 0,Y 321.557,Z 385.198,A -85,B 0,C 180,E1 -15803.965,E2 -15803.965} C_VEL
LIN {X 0,Y 322.782,Z 373.594,A -85,B 0,C 180,E1 -15804.913,E2 -15804.913} C_VEL
LIN {X 0,Y 322.715,Z 368.147,A -85,B 0,C 180,E1 -15805.326,E2 -15805.326} C_VEL
LIN {X 0,Y 320.777,Z 359.289,A -85,B 0,C 180,E1 -15806.049,E2 -15806.049} C_VEL
LIN {X 0,Y 318.701,Z 350.243,A -85,B 0,C 180,E1 -15806.659,E2 -15806.659} C_VEL
LIN {X 0,Y 318.347,Z 344.513,A -85,B 0,C 180,E1 -15806.887,E2 -15806.887} C_VEL
LIN {X 0,Y 320.585,Z 272.852,A -85,B 0,C 180,E1 -15808.62,E2 -15808.62} C_VEL
LIN {X 0,Y 318.812,Z 267.674,A -85,B 0,C 180,E1 -15808.944,E2 -15808.944} C_VEL
LIN {X 0,Y 312.852,Z 253.987,A -85,B 0,C 180,E1 -15809.975,E2 -15809.975} C_VEL
LIN {X 0,Y 306.836,Z 241.631,A -85,B 0,C 180,E1 -15811.065,E2 -15811.065} C_VEL
LIN {X 0,Y 305.482,Z 236.434,A -85,B 0,C 180,E1 -15812.974,E2 -15812.974} C_VEL
LIN {X 0,Y 305.481,Z 236.433,A -85,B 0,C 180,E1 -15815.546,E2 -15815.546} C_VEL
LIN {X 0,Y 305.495,Z 236.432,A -85,B 0,C 180,E1 -15819.823,E2 -15819.823} C_VEL
LIN {X 0,Y 305.552,Z 236.424,A -85,B 0,C 180,E1 -15822.611,E2 -15822.611} C_VEL
LIN {X 0,Y 305.63,Z 236.412,A -85,B 0,C 180,E1 -15825.357,E2 -15825.357} C_VEL
LIN {X 0,Y 305.62,Z 236.417,A -85,B 0,C 180,E1 -15829.407,E2 -15829.407} C_VEL
LIN {X 0,Y 305.755,Z 236.394,A -85,B 0,C 180,E1 -15832.081,E2 -15832.081} C_VEL
LIN {X 0,Y 305.662,Z 236.405,A -85,B 0,C 180,E1 -15834.731,E2 -15834.731} C_VEL
LIN {X 0,Y 305.943,Z 236.369,A -85,B 0,C 180,E1 -15838.691,E2 -15838.691} C_VEL
LIN {X 0,Y 305.941,Z 236.369,A -85,B 0,C 180,E1 -15841.324,E2 -15841.324} C_VEL
LIN {X 0,Y 305.799,Z 236.385,A -85,B 0,C 180,E1 -15846.606,E2 -15846.606} C_VEL
LIN {X 0,Y 305.691,Z 236.399,A -85,B 0,C 180,E1 -15849.268,E2 -15849.268} C_VEL
LIN {X 0,Y 305.584,Z 236.415,A -85,B 0,C 180,E1 -15853.303,E2 -15853.303} C_VEL
LIN {X 0,Y 305.552,Z 236.423,A -85,B 0,C 180,E1 -15856.029,E2 -15856.029} C_VEL
LIN {X 0,Y 305.485,Z 236.431,A -85,B 0,C 180,E1 -15860.194,E2 -15860.194} C_VEL
LIN {X 0,Y 305.451,Z 236.437,A -85,B 0,C 180,E1 -15864.473,E2 -15864.473} C_VEL
LIN {X 0,Y 305.446,Z 236.434,A -85,B 0,C 180,E1 -15867.405,E2 -15867.405} C_VEL
LIN {X 0,Y 305.421,Z 236.434,A -85,B 0,C 180,E1 -15870.42,E2 -15870.42} C_VEL
LIN {X 0,Y 305.473,Z 236.428,A -85,B 0,C 180,E1 -15874.083,E2 -15874.083} C_VEL
LIN {X 0,Y 305.46,Z 236.431,A -85,B 0,C 180,E1 -15876.748,E2 -15876.748} C_VEL
LIN {X 0,Y 305.406,Z 236.443,A -85,B 0,C 180,E1 -15880.591,E2 -15880.591} C_VEL
LIN {X 0,Y 305.4,Z 236.446,A -85,B 0,C 180,E1 -15884.491,E2 -15884.491} C_VEL
LIN {X 0,Y 305.401,Z 236.449,A -85,B 0,C 180,E1 -15888.138,E2 -15888.138} C_VEL
LIN {X 0,Y 305.441,Z 236.439,A -85,B 0,C 180,E1 -15891.594,E2 -15891.594} C_VEL
LIN {X 0,Y 305.522,Z 236.615,A -85,B 0,C 180,E1 -15894.896,E2 -15894.896} C_VEL
LIN {X 0,Y 308.455,Z 248.152,A -85,B 0,C 180,E1 -15898.78,E2 -15898.78} C_VEL
LIN {X 0,Y 310.541,Z 258.447,A -85,B 0,C 180,E1 -15901.97,E2 -15901.97} C_VEL
LIN {X 0,Y 310.878,Z 260.197,A -85,B 0,C 180,E1 -15902.483,E2 -15902.483} C_VEL
LIN {X 0,Y 313.042,Z 265.985,A -85,B 0,C 180,E1 -15902.891,E2 -15902.891} C_VEL
LIN {X 0,Y 317.292,Z 287.801,A -85,B 0,C 180,E1 -15903.958,E2 -15903.958} C_VEL
LIN {X 0,Y 319.726,Z 304.569,A -85,B 0,C 180,E1 -15904.662,E2 -15904.662} C_VEL
LIN {X 0,Y 317.714,Z 370.011,A -85,B 0,C 180,E1 -15906.276,E2 -15906.276} C_VEL
LIN {X 0,Y 316.659,Z 383.465,A -85,B 0,C 180,E1 -15906.844,E2 -15906.844} C_VEL
LIN {X 0,Y 315.331,Z 396.258,A -85,B 0,C 180,E1 -15907.649,E2 -15907.649} C_VEL
LIN {X 0,Y 313.806,Z 407.981,A -85,B 0,C 180,E1 -15908.659,E2 -15908.659} C_VEL
LIN {X 0,Y 312.051,Z 419.335,A -85,B 0,C 180,E1 -15909.913,E2 -15909.913} C_VEL
LIN {X 0,Y 310.348,Z 429.644,A -85,B 0,C 180,E1 -15911.346,E2 -15911.346} C_VEL
LIN {X 0,Y 308.801,Z 438.778,A -85,B 0,C 180,E1 -15912.93,E2 -15912.93} C_VEL
LIN {X 0,Y 307.351,Z 447.297,A -85,B 0,C 180,E1 -15914.755,E2 -15914.755} C_VEL
LIN {X 0,Y 305.92,Z 454.734,A -85,B 0,C 180,E1 -15916.719,E2 -15916.719} C_VEL
LIN {X 0,Y 304.919,Z 460.72,A -85,B 0,C 180,E1 -15918.702,E2 -15918.702} C_VEL
LIN {X 0,Y 304.246,Z 465.462,A -85,B 0,C 180,E1 -15920.695,E2 -15920.695} C_VEL
